C03575=1022.958,345.927,-141.680,171.455,48.856,159.616
C03576=1022.966,346.174,-141.717,171.462,48.856,159.617
C03577=1022.973,346.421,-141.753,171.468,48.855,159.618
C03578=1022.981,346.668,-141.790,171.475,48.854,159.618
C03579=1022.989,346.915,-141.828,171.483,48.853,159.619
C03580=1022.997,347.162,-141.865,171.489,48.852,159.620
C03581=1023.003,347.410,-141.902,171.496,48.851,159.621
C03582=1023.011,347.657,-141.939,171.502,48.850,159.622
C03583=1023.019,347.904,-141.976,171.510,48.849,159.623
C03584=1023.027,348.151,-142.013,171.517,48.848,159.623
C03585=1023.034,348.398,-142.051,171.524,48.848,159.624
C03586=1023.042,348.645,-142.087,171.530,48.847,159.625
C03587=1023.050,348.892,-142.125,171.538,48.846,159.626
C03588=1023.057,349.140,-142.163,171.545,48.845,159.627
C03589=1023.065,349.386,-142.200,171.551,48.845,159.628
C03590=1023.072,349.634,-142.237,171.559,48.844,159.629
C03591=1023.079,349.881,-142.275,171.566,48.843,159.629
C03592=1023.087,350.127,-142.312,171.573,48.843,159.630
C03593=1023.095,350.375,-142.349,171.580,48.842,159.631
C03594=1023.103,350.622,-142.387,171.587,48.841,159.632
C03595=1023.110,350.869,-142.424,171.594,48.840,159.633
C03596=1023.117,351.103,-142.460,171.601,48.840,159.634
C03597=1023.125,351.336,-142.495,171.607,48.839,159.635
C03598=1023.132,351.570,-142.532,171.614,48.838,159.635
C03599=1023.139,351.803,-142.567,171.621,48.838,159.636
C03600=1023.147,352.037,-142.602,171.628,48.838,159.637
C03601=1023.154,352.271,-142.638,171.635,48.837,159.638
C03602=1023.161,352.504,-142.673,171.641,48.836,159.639
C03603=1023.169,352.738,-142.709,171.648,48.836,159.640
C03604=1023.176,352.984,-142.747,171.656,48.835,159.641
C03605=1023.185,353.232,-142.784,171.662,48.834,159.642
C03606=1023.192,353.479,-142.822,171.669,48.834,159.643
C03607=1023.200,353.725,-142.860,171.677,48.833,159.644
C03608=1023.208,353.973,-142.897,171.684,48.832,159.644
C03609=1023.216,354.219,-142.935,171.692,48.832,159.646
C03610=1023.224,354.467,-142.973,171.699,48.831,159.646
C03611=1023.231,354.714,-143.012,171.707,48.831,159.648
C03612=1023.240,354.960,-143.049,171.714,48.830,159.648
C03613=1023.247,355.208,-143.087,171.721,48.830,159.649
C03614=1023.255,355.454,-143.125,171.728,48.829,159.650
C03615=1023.263,355.701,-143.164,171.735,48.829,159.651
C03616=1023.270,355.949,-143.201,171.743,48.828,159.652
C03617=1023.278,356.196,-143.240,171.750,48.828,159.653
C03618=1023.287,356.442,-143.278,171.758,48.827,159.654
C03619=1023.295,356.690,-143.316,171.765,48.827,159.655
C03620=1023.302,356.936,-143.354,171.773,48.827,159.656
C03621=1023.310,357.184,-143.392,171.780,48.826,159.657
C03622=1023.318,357.430,-143.431,171.788,48.826,159.658
C03623=1023.326,357.677,-143.469,171.795,48.825,159.659
C03624=1023.334,357.924,-143.508,171.803,48.824,159.660
C03625=1023.342,358.171,-143.546,171.810,48.824,159.661
C03626=1023.350,358.417,-143.584,171.818,48.824,159.663
C03627=1023.358,358.664,-143.622,171.825,48.824,159.664
C03628=1023.366,358.912,-143.661,171.833,48.824,159.665
C03629=1023.374,359.158,-143.699,171.840,48.823,159.666
C03630=1023.382,359.405,-143.738,171.848,48.823,159.667
C03631=1023.390,359.653,-143.776,171.855,48.823,159.668
C03632=1023.398,359.899,-143.815,171.863,48.822,159.669
C03633=1023.406,360.146,-143.853,171.870,48.822,159.670
C03634=1023.414,360.394,-143.892,171.878,48.822,159.671
C03635=1023.422,360.639,-143.931,171.885,48.822,159.672
C03636=1023.429,360.887,-143.970,171.893,48.821,159.673
C03637=1023.437,361.134,-144.009,171.900,48.821,159.674
C03638=1023.445,361.380,-144.048,171.908,48.821,159.675
C03639=1023.453,361.627,-144.086,171.916,48.820,159.676
C03640=1023.462,361.874,-144.126,171.924,48.820,159.677
C03641=1023.470,362.121,-144.164,171.932,48.821,159.679
C03642=1023.477,362.367,-144.204,171.939,48.821,159.680
C03643=1023.485,362.615,-144.242,171.947,48.820,159.681
C03644=1023.494,362.861,-144.282,171.955,48.820,159.682
C03645=1023.502,363.108,-144.320,171.963,48.820,159.683
C03646=1023.510,363.355,-144.360,171.971,48.820,159.684
C03647=1023.517,363.602,-144.398,171.978,48.820,159.685
C03648=1023.526,363.848,-144.438,171.986,48.819,159.687
C03649=1023.534,364.095,-144.477,171.994,48.820,159.688
C03650=1023.542,364.342,-144.516,172.001,48.820,159.689
C03651=1023.551,364.589,-144.555,172.009,48.819,159.690
C03652=1023.558,364.836,-144.595,172.018,48.819,159.691
C03653=1023.567,365.083,-144.634,172.025,48.819,159.692
C03654=1023.575,365.330,-144.673,172.033,48.820,159.694
C03655=1023.583,365.576,-144.712,172.041,48.819,159.695
C03656=1023.591,365.813,-144.750,172.049,48.819,159.696
C03657=1023.599,366.049,-144.788,172.057,48.819,159.697
C03658=1023.608,366.287,-144.825,172.064,48.819,159.698
C03659=1023.615,366.524,-144.863,172.072,48.819,159.700
C03660=1023.623,366.761,-144.901,172.080,48.819,159.701
C03661=1023.631,366.998,-144.940,172.088,48.820,159.702
C03662=1023.639,367.235,-144.977,172.095,48.820,159.703
C03663=1023.647,367.471,-145.015,172.103,48.819,159.704
C03664=1023.656,367.719,-145.055,172.111,48.820,159.705
C03665=1023.664,367.965,-145.094,172.119,48.820,159.707
C03666=1023.673,368.212,-145.134,172.127,48.819,159.708
C03667=1023.680,368.459,-145.174,172.135,48.820,159.709
C03668=1023.689,368.705,-145.213,172.144,48.820,159.710
C03669=1023.697,368.952,-145.253,172.151,48.820,159.712
C03670=1023.705,369.198,-145.293,172.160,48.821,159.713
C03671=1023.713,369.445,-145.333,172.168,48.821,159.714
C03672=1023.722,369.693,-145.372,172.177,48.821,159.716
C03673=1023.730,369.939,-145.413,172.185,48.821,159.717
C03674=1023.739,370.185,-145.452,172.192,48.822,159.718
C03675=1023.747,370.432,-145.493,172.201,48.822,159.719
C03676=1023.755,370.678,-145.532,172.209,48.822,159.721
C03677=1023.764,370.925,-145.573,172.218,48.822,159.722
C03678=1023.772,371.172,-145.613,172.226,48.823,159.723
C03679=1023.780,371.418,-145.653,172.235,48.823,159.725
C03680=1023.789,371.665,-145.693,172.243,48.823,159.726
C03681=1023.797,371.912,-145.734,172.250,48.824,159.727
C03682=1023.806,372.158,-145.774,172.259,48.824,159.729
C03683=1023.814,372.405,-145.814,172.267,48.824,159.730
C03684=1023.822,372.652,-145.855,172.276,48.825,159.731
C03685=1023.831,372.898,-145.895,172.284,48.825,159.733
C03686=1023.839,373.145,-145.935,172.293,48.825,159.734
C03687=1023.848,373.391,-145.975,172.301,48.825,159.735
C03688=1023.856,373.637,-146.016,172.310,48.826,159.737
C03689=1023.866,373.884,-146.056,172.319,48.826,159.738
C03690=1023.874,374.130,-146.097,172.327,48.826,159.740
C03691=1023.883,374.377,-146.137,172.336,48.827,159.741
C03692=1023.891,374.623,-146.178,172.344,48.827,159.742
C03693=1023.900,374.870,-146.218,172.353,48.828,159.744
C03694=1023.908,375.117,-146.258,172.361,48.828,159.745
C03695=1023.917,375.364,-146.298,172.370,48.829,159.747
C03696=1023.926,375.609,-146.340,172.379,48.829,159.748
C03697=1023.935,375.856,-146.380,172.387,48.830,159.750
C03698=1023.943,376.102,-146.421,172.396,48.830,159.751
C03699=1023.952,376.349,-146.462,172.405,48.831,159.752
C03700=1023.961,376.596,-146.502,172.413,48.831,159.754
C03701=1023.969,376.842,-146.543,172.422,48.832,159.755
C03702=1023.978,377.089,-146.585,172.431,48.833,159.757
C03703=1023.987,377.336,-146.626,172.439,48.833,159.758
C03704=1023.995,377.582,-146.666,172.448,48.834,159.760
C03705=1024.004,377.828,-146.707,172.457,48.835,159.761
C03706=1024.013,378.074,-146.748,172.466,48.835,159.763
C03707=1024.021,378.320,-146.790,172.475,48.836,159.764
C03708=1024.030,378.567,-146.831,172.484,48.837,159.766
C03709=1024.038,378.813,-146.872,172.493,48.838,159.767
C03710=1024.047,379.060,-146.913,172.501,48.838,159.769
C03711=1024.056,379.306,-146.955,172.510,48.839,159.770
C03712=1024.065,379.553,-146.997,172.519,48.840,159.772
C03713=1024.073,379.799,-147.037,172.528,48.841,159.773
C03714=1024.083,380.045,-147.078,172.538,48.841,159.775
C03715=1024.092,380.292,-147.120,172.546,48.842,159.776
C03716=1024.100,380.541,-147.162,172.555,48.843,159.778
C03717=1024.109,380.790,-147.203,172.564,48.843,159.779
C03718=1024.118,381.039,-147.246,172.574,48.844,159.781
C03719=1024.127,381.288,-147.287,172.583,48.845,159.783
C03720=1024.136,381.535,-147.329,172.592,48.846,159.784
C03721=1024.145,381.781,-147.371,172.601,48.846,159.786
C03722=1024.154,382.027,-147.412,172.610,48.847,159.787
C03723=1024.163,382.274,-147.454,172.619,48.849,159.789
C03724=1024.172,382.520,-147.496,172.628,48.849,159.791
C03725=1024.181,382.766,-147.537,172.638,48.850,159.792
C03726=1024.190,383.013,-147.579,172.647,48.851,159.794
C03727=1024.199,383.259,-147.620,172.656,48.852,159.795
C03728=1024.208,383.505,-147.662,172.666,48.852,159.797
C03729=1024.217,383.752,-147.704,172.675,48.854,159.799
C03730=1024.226,383.998,-147.745,172.684,48.854,159.800
C03731=1024.235,384.244,-147.788,172.694,48.855,159.802
C03732=1024.244,384.490,-147.830,172.702,48.856,159.804
C03733=1024.253,384.737,-147.871,172.713,48.857,159.805
C03734=1024.263,384.983,-147.913,172.722,48.859,159.807
C03735=1024.273,385.229,-147.955,172.730,48.859,159.809
C03736=1024.282,385.475,-147.997,172.741,48.860,159.810
C03737=1024.290,385.722,-148.039,172.749,48.861,159.812
C03738=1024.300,385.968,-148.081,172.760,48.862,159.814
C03739=1024.309,386.215,-148.123,172.769,48.863,159.816
C03740=1024.318,386.460,-148.166,172.779,48.864,159.817
C03741=1024.327,386.706,-148.209,172.788,48.866,159.819
C03742=1024.336,386.953,-148.250,172.797,48.867,159.821
C03743=1024.346,387.199,-148.293,172.807,48.868,159.822
C03744=1024.355,387.445,-148.336,172.816,48.869,159.824
C03745=1024.364,387.691,-148.377,172.826,48.870,159.826
C03746=1024.373,387.937,-148.420,172.835,48.871,159.828
C03747=1024.383,388.183,-148.463,172.845,48.872,159.829
C03748=1024.391,388.430,-148.506,172.856,48.873,159.831
C03749=1024.401,388.676,-148.548,172.865,48.875,159.833
C03750=1024.411,388.922,-148.591,172.875,48.876,159.835
C03751=1024.420,389.167,-148.633,172.884,48.877,159.837
C03752=1024.429,389.414,-148.677,172.894,48.878,159.838
C03753=1024.438,389.660,-148.719,172.904,48.880,159.840
C03754=1024.448,389.906,-148.762,172.914,48.881,159.842
C03755=1024.457,390.152,-148.804,172.924,48.882,159.844
C03756=1024.466,390.398,-148.847,172.933,48.884,159.846
C03757=1024.476,390.645,-148.890,172.944,48.885,159.848
C03758=1024.485,390.890,-148.933,172.954,48.886,159.849
C03759=1024.494,391.137,-148.977,172.963,48.888,159.851
C03760=1024.504,391.383,-149.019,172.974,48.889,159.853
C03761=1024.513,391.629,-149.062,172.984,48.890,159.855
C03762=1024.523,391.875,-149.106,172.993,48.892,159.857
C03763=1024.532,392.121,-149.148,173.003,48.893,159.859
C03764=1024.542,392.367,-149.191,173.014,48.895,159.861
C03765=1024.551,392.613,-149.235,173.023,48.897,159.863
C03766=1024.560,392.859,-149.278,173.034,48.897,159.864
C03767=1024.571,393.105,-149.321,173.044,48.899,159.866
C03768=1024.580,393.351,-149.365,173.055,48.901,159.869
C03769=1024.589,393.597,-149.408,173.065,48.902,159.870
C03770=1024.599,393.843,-149.452,173.074,48.903,159.872
C03771=1024.609,394.089,-149.495,173.085,48.905,159.874
C03772=1024.617,394.335,-149.538,173.095,48.907,159.876
C03773=1024.627,394.580,-149.582,173.106,48.908,159.878
C03774=1024.637,394.827,-149.626,173.116,48.910,159.880
C03775=1024.647,395.072,-149.670,173.126,48.912,159.882
C03776=1024.658,395.359,-149.720,173.139,48.913,159.885
C03777=1024.669,395.643,-149.771,173.150,48.915,159.887
C03778=1024.681,395.930,-149.821,173.162,48.917,159.889
C03779=1024.692,396.216,-149.873,173.174,48.919,159.892
C03780=1024.702,396.461,-149.917,173.185,48.921,159.894
C03781=1024.711,396.708,-149.961,173.195,48.922,159.896
C03782=1024.721,396.953,-150.004,173.206,48.924,159.898
C03783=1024.731,397.199,-150.048,173.216,48.925,159.900
C03784=1024.741,397.445,-150.093,173.227,48.927,159.902
C03785=1024.751,397.691,-150.137,173.238,48.929,159.904
C03786=1024.761,397.937,-150.180,173.248,48.931,159.906
C03787=1024.770,398.183,-150.224,173.259,48.933,159.908
C03788=1024.781,398.428,-150.269,173.270,48.934,159.910
C03789=1024.790,398.674,-150.313,173.281,48.936,159.912
C03790=1024.800,398.920,-150.357,173.291,48.938,159.914
C03791=1024.810,399.165,-150.401,173.302,48.940,159.917
C03792=1024.820,399.411,-150.446,173.312,48.941,159.919
C03793=1024.830,399.658,-150.490,173.324,48.943,159.921
C03794=1024.840,399.903,-150.534,173.335,48.945,159.923
C03795=1024.850,400.149,-150.579,173.346,48.947,159.925
C03796=1024.860,400.394,-150.624,173.357,48.949,159.927
C03797=1024.869,400.640,-150.668,173.367,48.951,159.929
C03798=1024.880,400.886,-150.713,173.378,48.953,159.932
C03799=1024.890,401.132,-150.758,173.389,48.955,159.934
C03800=1024.899,401.377,-150.802,173.401,48.956,159.936
C03801=1024.909,401.623,-150.847,173.411,48.959,159.938
C03802=1024.919,401.869,-150.892,173.422,48.961,159.940
C03803=1024.929,402.114,-150.937,173.433,48.963,159.943
C03804=1024.940,402.360,-150.982,173.445,48.964,159.945
C03805=1024.950,402.606,-151.027,173.456,48.967,159.947
C03806=1024.960,402.851,-151.072,173.467,48.969,159.950
C03807=1024.970,403.097,-151.117,173.478,48.971,159.952
C03808=1024.980,403.342,-151.162,173.490,48.973,159.954
C03809=1024.990,403.588,-151.207,173.501,48.975,159.956
C03810=1025.000,403.834,-151.252,173.512,48.978,159.959
C03811=1025.010,404.079,-151.298,173.524,48.980,159.961
C03812=1025.020,404.325,-151.343,173.535,48.982,159.963
C03813=1025.030,404.571,-151.388,173.547,48.984,159.966
C03814=1025.041,404.816,-151.434,173.558,48.986,159.968
C03815=1025.051,405.063,-151.479,173.569,48.988,159.970
C03816=1025.062,405.307,-151.524,173.581,48.990,159.973
C03817=1025.072,405.553,-151.569,173.592,48.992,159.975
C03818=1025.083,405.799,-151.615,173.604,48.995,159.977
C03819=1025.093,406.044,-151.661,173.615,48.997,159.980
C03820=1025.103,406.290,-151.706,173.627,48.999,159.982
C03821=1025.114,406.536,-151.752,173.638,49.002,159.985
C03822=1025.124,406.781,-151.798,173.651,49.004,159.987
C03823=1025.134,407.026,-151.843,173.662,49.006,159.989
C03824=1025.145,407.272,-151.888,173.674,49.008,159.992
C03825=1025.155,407.518,-151.934,173.686,49.011,159.994
C03826=1025.166,407.763,-151.980,173.697,49.013,159.997
C03827=1025.176,408.009,-152.026,173.709,49.016,159.999
C03828=1025.188,408.254,-152.071,173.722,49.018,160.002
C03829=1025.198,408.500,-152.117,173.733,49.020,160.004
C03830=1025.209,408.746,-152.163,173.745,49.023,160.007
C03831=1025.220,408.991,-152.209,173.757,49.025,160.009
C03832=1025.230,409.237,-152.255,173.770,49.027,160.012
C03833=1025.241,409.482,-152.301,173.781,49.030,160.014
C03834=1025.252,409.727,-152.347,173.793,49.032,160.017
C03835=1025.263,409.973,-152.393,173.806,49.035,160.019
C03836=1025.275,410.282,-152.452,173.821,49.038,160.022
C03837=1025.289,410.590,-152.511,173.836,49.041,160.026
C03838=1025.302,410.898,-152.568,173.851,49.044,160.029
C03839=1025.316,411.206,-152.627,173.867,49.048,160.032
C03840=1025.326,411.451,-152.673,173.879,49.050,160.035
C03841=1025.337,411.697,-152.721,173.891,49.053,160.037
C03842=1025.348,411.942,-152.767,173.904,49.056,160.040
C03843=1025.359,412.188,-152.813,173.916,49.058,160.043
C03844=1025.370,412.433,-152.860,173.929,49.061,160.045
C03845=1025.380,412.679,-152.907,173.941,49.063,160.048
C03846=1025.391,412.924,-152.954,173.954,49.066,160.051
C03847=1025.402,413.169,-153.001,173.966,49.068,160.053
C03848=1025.414,413.414,-153.048,173.979,49.071,160.056
C03849=1025.424,413.660,-153.095,173.992,49.074,160.059
C03850=1025.435,413.905,-153.141,174.004,49.077,160.062
C03851=1025.446,414.150,-153.188,174.017,49.080,160.064
C03852=1025.457,414.395,-153.235,174.029,49.082,160.067
C03853=1025.468,414.641,-153.283,174.042,49.085,160.070
C03854=1025.479,414.886,-153.329,174.055,49.088,160.072
C03855=1025.491,415.131,-153.377,174.069,49.091,160.075
C03856=1025.502,415.377,-153.424,174.081,49.094,160.078
C03857=1025.513,415.622,-153.471,174.094,49.097,160.081
C03858=1025.524,415.868,-153.518,174.106,49.099,160.084
C03859=1025.535,416.113,-153.566,174.119,49.103,160.087
C03860=1025.546,416.358,-153.613,174.133,49.105,160.089
C03861=1025.557,416.604,-153.661,174.146,49.108,160.092
C03862=1025.569,416.849,-153.709,174.159,49.111,160.095
C03863=1025.579,417.094,-153.756,174.173,49.114,160.098
C03864=1025.591,417.339,-153.804,174.185,49.117,160.101
C03865=1025.602,417.584,-153.852,174.198,49.120,160.104
C03866=1025.614,417.829,-153.900,174.212,49.123,160.107
C03867=1025.625,418.074,-153.948,174.225,49.127,160.110
C03868=1025.636,418.320,-153.995,174.238,49.129,160.112
C03869=1025.647,418.565,-154.043,174.252,49.132,160.115
C03870=1025.659,418.810,-154.091,174.265,49.136,160.118
C03871=1025.670,419.056,-154.139,174.279,49.139,160.121
C03872=1025.682,419.300,-154.188,174.292,49.142,160.124
C03873=1025.693,419.545,-154.236,174.306,49.145,160.127
C03874=1025.705,419.790,-154.284,174.320,49.148,160.130
C03875=1025.716,420.036,-154.332,174.333,49.151,160.133
C03876=1025.728,420.281,-154.380,174.347,49.155,160.136
C03877=1025.740,420.526,-154.429,174.360,49.158,160.139
C03878=1025.751,420.771,-154.476,174.374,49.161,160.142
C03879=1025.762,421.016,-154.525,174.388,49.164,160.145
C03880=1025.775,421.260,-154.573,174.401,49.167,160.149
C03881=1025.786,421.506,-154.621,174.415,49.170,160.152
C03882=1025.798,421.751,-154.670,174.430,49.174,160.155
C03883=1025.810,421.996,-154.718,174.444,49.177,160.158
C03884=1025.821,422.241,-154.767,174.458,49.180,160.161
C03885=1025.833,422.485,-154.816,174.471,49.184,160.164
C03886=1025.845,422.731,-154.865,174.485,49.187,160.167
C03887=1025.857,422.976,-154.914,174.500,49.190,160.170
C03888=1025.868,423.220,-154.963,174.514,49.194,160.174
C03889=1025.881,423.466,-155.012,174.528,49.197,160.177
C03890=1025.892,423.710,-155.061,174.542,49.200,160.180
C03891=1025.903,423.955,-155.110,174.557,49.204,160.183
C03892=1025.915,424.200,-155.159,174.571,49.207,160.186
C03893=1025.928,424.445,-155.208,174.585,49.211,160.190
C03894=1025.940,424.690,-155.257,174.600,49.215,160.193
C03895=1025.951,424.935,-155.306,174.615,49.218,160.196
C03896=1025.967,425.254,-155.371,174.633,49.223,160.201
C03897=1025.982,425.573,-155.435,174.652,49.227,160.205
C03898=1025.998,425.892,-155.499,174.671,49.232,160.209
C03899=1026.014,426.211,-155.563,174.691,49.236,160.214
C03900=1026.027,426.455,-155.613,174.706,49.240,160.217
C03901=1026.039,426.701,-155.663,174.720,49.244,160.220
C03902=1026.050,426.945,-155.713,174.735,49.248,160.224
C03903=1026.063,427.190,-155.763,174.750,49.251,160.227
C03904=1026.075,427.435,-155.813,174.765,49.255,160.230
C03905=1026.087,427.679,-155.863,174.780,49.259,160.234
C03906=1026.099,427.924,-155.913,174.795,49.262,160.237
C03907=1026.111,428.168,-155.963,174.810,49.266,160.241
C03908=1026.124,428.413,-156.013,174.825,49.270,160.244
C03909=1026.136,428.658,-156.063,174.840,49.274,160.248
C03910=1026.148,428.903,-156.113,174.855,49.278,160.251
C03911=1026.160,429.148,-156.163,174.871,49.281,160.255
C03912=1026.173,429.393,-156.213,174.886,49.285,160.258
C03913=1026.185,429.637,-156.264,174.901,49.289,160.262
C03914=1026.198,429.882,-156.314,174.918,49.293,160.266
C03915=1026.210,430.126,-156.365,174.932,49.297,160.269
C03916=1026.223,430.371,-156.415,174.948,49.300,160.273
C03917=1026.235,430.615,-156.465,174.963,49.305,160.276
C03918=1026.248,430.860,-156.516,174.979,49.308,160.280
C03919=1026.261,431.105,-156.567,174.995,49.312,160.284
C03920=1026.273,431.349,-156.617,175.011,49.316,160.287
C03921=1026.286,431.594,-156.668,175.027,49.320,160.291
C03922=1026.298,431.838,-156.719,175.042,49.324,160.294
C03923=1026.312,432.083,-156.770,175.058,49.329,160.298
C03924=1026.324,432.327,-156.820,175.074,49.333,160.302
C03925=1026.337,432.572,-156.871,175.090,49.337,160.306
C03926=1026.350,432.817,-156.922,175.107,49.341,160.309
C03927=1026.363,433.061,-156.973,175.123,49.345,160.313
C03928=1026.376,433.306,-157.024,175.139,49.349,160.317
C03929=1026.389,433.550,-157.076,175.155,49.353,160.321
C03930=1026.402,433.794,-157.127,175.171,49.357,160.324
C03931=1026.414,434.038,-157.178,175.188,49.361,160.328
C03932=1026.428,434.283,-157.229,175.204,49.365,160.332
C03933=1026.441,434.528,-157.281,175.220,49.370,160.336
C03934=1026.453,434.771,-157.333,175.237,49.374,160.340
C03935=1026.466,435.016,-157.384,175.254,49.378,160.344
C03936=1026.480,435.261,-157.436,175.270,49.382,160.348
C03937=1026.493,435.505,-157.487,175.287,49.387,160.352
C03938=1026.506,435.749,-157.538,175.304,49.391,160.356
C03939=1026.519,435.994,-157.591,175.321,49.396,160.360
C03940=1026.532,436.237,-157.643,175.337,49.400,160.363
C03941=1026.545,436.482,-157.694,175.354,49.404,160.367
C03942=1026.559,436.726,-157.746,175.371,49.408,160.371
C03943=1026.572,436.970,-157.799,175.389,49.413,160.376
C03944=1026.585,437.215,-157.851,175.405,49.417,160.380
C03945=1026.599,437.459,-157.903,175.423,49.422,160.384
C03946=1026.612,437.703,-157.954,175.439,49.426,160.388
C03947=1026.625,437.947,-158.008,175.457,49.431,160.392
C03948=1026.639,438.192,-158.060,175.475,49.435,160.396
C03949=1026.652,438.436,-158.111,175.491,49.439,160.400
C03950=1026.666,438.680,-158.165,175.509,49.444,160.404
C03951=1026.679,438.924,-158.217,175.527,49.449,160.409
C03952=1026.693,439.168,-158.269,175.543,49.453,160.413
C03953=1026.706,439.412,-158.322,175.561,49.458,160.417
C03954=1026.720,439.656,-158.374,175.579,49.462,160.421
C03955=1026.734,439.900,-158.427,175.597,49.467,160.425
C03956=1026.747,440.144,-158.480,175.615,49.472,160.430
C03957=1026.760,440.390,-158.533,175.633,49.476,160.434
C03958=1026.775,440.634,-158.586,175.651,49.481,160.438
C03959=1026.789,440.879,-158.640,175.669,49.486,160.442
C03960=1026.801,441.107,-158.689,175.686,49.490,160.447
C03961=1026.815,441.334,-158.738,175.703,49.495,160.451
C03962=1026.828,441.561,-158.788,175.720,49.499,160.455
C03963=1026.840,441.790,-158.838,175.736,49.503,160.459
C03964=1026.853,442.017,-158.888,175.754,49.508,160.463
C03965=1026.867,442.244,-158.937,175.771,49.512,160.467
C03966=1026.880,442.472,-158.987,175.789,49.517,160.471
C03967=1026.893,442.700,-159.036,175.805,49.521,160.475
C03968=1026.908,442.942,-159.089,175.823,49.526,160.480
C03969=1026.922,443.185,-159.142,175.842,49.530,160.484
C03970=1026.938,443.429,-159.194,175.862,49.535,160.489
C03971=1026.954,443.673,-159.245,175.879,49.540,160.493
C03972=1026.971,443.916,-159.297,175.899,49.544,160.497
C03973=1026.987,444.160,-159.347,175.918,49.548,160.502
C03974=1027.005,444.403,-159.398,175.937,49.553,160.506
C03975=1027.022,444.648,-159.448,175.956,49.557,160.511
C03976=1027.041,444.892,-159.498,175.975,49.561,160.515
C03977=1027.060,445.136,-159.547,175.994,49.565,160.519
C03978=1027.079,445.380,-159.595,176.013,49.569,160.524
C03979=1027.098,445.624,-159.644,176.033,49.573,160.528
C03980=1027.118,445.869,-159.692,176.052,49.577,160.532
C03981=1027.138,446.113,-159.739,176.072,49.581,160.537
C03982=1027.159,446.357,-159.787,176.092,49.585,160.541
C03983=1027.181,446.601,-159.834,176.112,49.588,160.545
C03984=1027.203,446.845,-159.881,176.132,49.592,160.550
C03985=1027.225,447.091,-159.927,176.151,49.596,160.554
C03986=1027.248,447.335,-159.972,176.172,49.599,160.559
C03987=1027.272,447.580,-160.017,176.192,49.603,160.563
C03988=1027.295,447.825,-160.062,176.212,49.606,160.567
C03989=1027.319,448.069,-160.107,176.232,49.609,160.571
C03990=1027.345,448.315,-160.151,176.253,49.612,160.576
C03991=1027.369,448.559,-160.195,176.274,49.615,160.580
C03992=1027.395,448.804,-160.239,176.295,49.619,160.585
C03993=1027.421,449.049,-160.281,176.315,49.621,160.589
C03994=1027.447,449.295,-160.323,176.336,49.624,160.593
C03995=1027.475,449.539,-160.365,176.357,49.628,160.597
C03996=1027.502,449.785,-160.407,176.377,49.630,160.602
C03997=1027.530,450.030,-160.449,176.399,49.633,160.606
C03998=1027.559,450.275,-160.490,176.419,49.636,160.610
C03999=1027.587,450.521,-160.531,176.441,49.638,160.615
C04000=1027.617,450.766,-160.571,176.462,49.641,160.619
C04001=1027.646,451.012,-160.611,176.483,49.644,160.623
C04002=1027.677,451.257,-160.650,176.504,49.647,160.628
C04003=1027.707,451.502,-160.689,176.526,49.649,160.632
C04004=1027.738,451.748,-160.728,176.548,49.651,160.636
C04005=1027.771,451.994,-160.765,176.570,49.653,160.640
C04006=1027.802,452.240,-160.804,176.591,49.656,160.645
C04007=1027.835,452.485,-160.841,176.614,49.658,160.649
C04008=1027.868,452.731,-160.878,176.635,49.660,160.653
C04009=1027.902,452.977,-160.914,176.658,49.662,160.658
C04010=1027.935,453.222,-160.950,176.680,49.664,160.662
C04011=1027.971,453.468,-160.987,176.703,49.666,160.666
C04012=1028.005,453.714,-161.021,176.725,49.668,160.671
C04013=1028.040,453.960,-161.057,176.747,49.670,160.675
C04014=1028.076,454.206,-161.091,176.770,49.672,160.679
C04015=1028.113,454.451,-161.125,176.792,49.674,160.683
C04016=1027.838,454.527,-161.463,176.795,49.734,160.703
C04017=1027.801,454.282,-161.428,176.773,49.732,160.699
C04018=1027.765,454.036,-161.394,176.749,49.731,160.694
C04019=1027.730,453.790,-161.359,176.727,49.729,160.690
C04020=1027.695,453.544,-161.324,176.705,49.727,160.686
C04021=1027.660,453.298,-161.289,176.682,49.725,160.681
C04022=1027.626,453.053,-161.252,176.660,49.723,160.677
C04023=1027.593,452.807,-161.215,176.638,49.722,160.673
C04024=1027.560,452.561,-161.179,176.616,49.719,160.669
C04025=1027.527,452.316,-161.142,176.594,49.717,160.664
C04026=1027.494,452.070,-161.104,176.572,49.715,160.660
C04027=1027.463,451.824,-161.066,176.550,49.713,160.656
C04028=1027.431,451.578,-161.028,176.528,49.711,160.652
C04029=1027.400,451.334,-160.988,176.506,49.708,160.647
C04030=1027.370,451.088,-160.950,176.485,49.706,160.643
C04031=1027.340,450.842,-160.910,176.463,49.703,160.639
C04032=1027.310,450.596,-160.870,176.442,49.701,160.634
C04033=1027.281,450.351,-160.829,176.421,49.699,160.630
C04034=1027.253,450.106,-160.789,176.400,49.695,160.626
C04035=1027.224,449.861,-160.748,176.378,49.693,160.621
C04036=1027.197,449.616,-160.706,176.358,49.690,160.617
C04037=1027.170,449.370,-160.664,176.336,49.687,160.613
C04038=1027.143,449.126,-160.622,176.316,49.685,160.609
C04039=1027.117,448.880,-160.579,176.295,49.681,160.604
C04040=1027.091,448.635,-160.535,176.274,49.679,160.600
C04041=1027.065,448.390,-160.492,176.254,49.676,160.596
C04042=1027.041,448.145,-160.449,176.233,49.672,160.591
C04043=1027.016,447.900,-160.404,176.213,49.670,160.587
C04044=1026.992,447.656,-160.359,176.193,49.666,160.583
C04045=1026.969,447.411,-160.314,176.172,49.663,160.578
C04046=1026.945,447.166,-160.268,176.152,49.659,160.574
C04047=1026.923,446.921,-160.223,176.132,49.656,160.570
C04048=1026.902,446.677,-160.176,176.112,49.653,160.565
C04049=1026.880,446.432,-160.129,176.092,49.649,160.561
C04050=1026.858,446.187,-160.082,176.072,49.646,160.557
C04051=1026.838,445.944,-160.035,176.052,49.642,160.552
C04052=1026.817,445.699,-159.987,176.033,49.638,160.548
C04053=1026.798,445.455,-159.939,176.013,49.634,160.544
C04054=1026.778,445.210,-159.890,175.994,49.630,160.539
C04055=1026.759,444.967,-159.841,175.975,49.626,160.535
C04056=1026.741,444.723,-159.791,175.956,49.622,160.531
C04057=1026.723,444.479,-159.742,175.936,49.618,160.526
C04058=1026.705,444.234,-159.692,175.917,49.614,160.522
C04059=1026.688,443.991,-159.641,175.898,49.610,160.517
C04060=1026.671,443.748,-159.590,175.879,49.606,160.513
C04061=1026.655,443.503,-159.539,175.860,49.601,160.508
C04062=1026.639,443.260,-159.486,175.842,49.597,160.504
C04063=1026.625,443.017,-159.434,175.823,49.592,160.500
C04064=1026.610,442.774,-159.381,175.804,49.587,160.495
C04065=1026.595,442.531,-159.329,175.786,49.583,160.491
C04066=1026.581,442.287,-159.275,175.767,49.578,160.486
C04067=1026.567,442.043,-159.223,175.749,49.573,160.482
C04068=1026.553,441.800,-159.169,175.730,49.569,160.478
C04069=1026.540,441.576,-159.121,175.714,49.565,160.474
C04070=1026.527,441.353,-159.072,175.697,49.561,160.470
C04071=1026.515,441.129,-159.024,175.681,49.556,160.466
C04072=1026.502,440.905,-158.975,175.664,49.552,160.462
C04073=1026.489,440.681,-158.926,175.648,49.547,160.458
C04074=1026.477,440.458,-158.877,175.630,49.544,160.454
C04075=1026.464,440.234,-158.829,175.614,49.540,160.450
C04076=1026.452,440.011,-158.781,175.597,49.535,160.446
C04077=1026.438,439.766,-158.727,175.580,49.531,160.442
C04078=1026.424,439.522,-158.675,175.563,49.526,160.438
C04079=1026.411,439.278,-158.623,175.545,49.521,160.433
C04080=1026.397,439.034,-158.570,175.527,49.517,160.429
C04081=1026.384,438.790,-158.517,175.509,49.513,160.425
C04082=1026.370,438.546,-158.465,175.492,49.508,160.421
C04083=1026.357,438.302,-158.412,175.474,49.504,160.417
C04084=1026.343,438.057,-158.360,175.457,49.499,160.413
C04085=1026.329,437.813,-158.308,175.440,49.495,160.408
C04086=1026.316,437.569,-158.256,175.422,49.491,160.404
C04087=1026.303,437.325,-158.203,175.405,49.486,160.400
C04088=1026.290,437.081,-158.151,175.388,49.482,160.396
C04089=1026.276,436.837,-158.099,175.371,49.478,160.392
C04090=1026.263,436.592,-158.047,175.354,49.473,160.388
C04091=1026.249,436.348,-157.996,175.337,49.469,160.384
C04092=1026.236,436.104,-157.943,175.320,49.465,160.380
C04093=1026.219,435.783,-157.875,175.298,49.459,160.375
C04094=1026.202,435.462,-157.807,175.276,49.454,160.370
C04095=1026.184,435.142,-157.740,175.254,49.449,160.365
C04096=1026.168,434.821,-157.673,175.233,49.443,160.360
C04097=1026.154,434.577,-157.621,175.215,49.439,160.356
C04098=1026.142,434.332,-157.569,175.199,49.435,160.352
C04099=1026.129,434.088,-157.517,175.183,49.431,160.348
C04100=1026.116,433.843,-157.466,175.166,49.426,160.344
C04101=1026.103,433.599,-157.415,175.150,49.422,160.340
C04102=1026.089,433.355,-157.364,175.134,49.418,160.337
C04103=1026.077,433.111,-157.313,175.117,49.414,160.333
C04104=1026.064,432.866,-157.262,175.101,49.410,160.329
C04105=1026.051,432.621,-157.211,175.085,49.406,160.325
C04106=1026.038,432.377,-157.160,175.069,49.402,160.322
C04107=1026.025,432.132,-157.109,175.053,49.399,160.318
C04108=1026.013,431.888,-157.059,175.038,49.394,160.314
C04109=1026.000,431.643,-157.008,175.021,49.390,160.311
C04110=1025.988,431.399,-156.957,175.006,49.387,160.307
C04111=1025.974,431.154,-156.906,174.990,49.383,160.303
C04112=1025.962,430.909,-156.856,174.974,49.379,160.300
C04113=1025.949,430.665,-156.805,174.958,49.375,160.296
C04114=1025.937,430.420,-156.755,174.943,49.371,160.292
C04115=1025.924,430.176,-156.704,174.927,49.368,160.289
C04116=1025.912,429.931,-156.654,174.911,49.364,160.285
C04117=1025.900,429.687,-156.604,174.896,49.360,160.282
C04118=1025.887,429.442,-156.553,174.880,49.356,160.278
C04119=1025.875,429.198,-156.503,174.865,49.353,160.275
C04120=1025.863,428.953,-156.453,174.850,49.349,160.271
C04121=1025.850,428.708,-156.403,174.834,49.345,160.268
C04122=1025.837,428.464,-156.353,174.819,49.341,160.264
C04123=1025.825,428.219,-156.302,174.804,49.338,160.261
C04124=1025.812,427.974,-156.252,174.789,49.334,160.257
C04125=1025.800,427.730,-156.202,174.773,49.330,160.254
C04126=1025.788,427.484,-156.153,174.759,49.327,160.250
C04127=1025.776,427.240,-156.103,174.743,49.323,160.247
C04128=1025.764,426.995,-156.053,174.729,49.320,160.244
C04129=1025.752,426.750,-156.003,174.714,49.316,160.240
C04130=1025.740,426.506,-155.953,174.699,49.312,160.237
C04131=1025.728,426.261,-155.904,174.684,49.309,160.233
C04132=1025.716,426.016,-155.854,174.669,49.305,160.230
C04133=1025.704,425.770,-155.804,174.654,49.302,160.227
C04134=1025.692,425.526,-155.755,174.640,49.298,160.223
C04135=1025.679,425.281,-155.706,174.625,49.295,160.220
C04136=1025.667,425.036,-155.656,174.610,49.292,160.217
C04137=1025.656,424.791,-155.607,174.596,49.288,160.214
C04138=1025.643,424.546,-155.557,174.582,49.285,160.210
C04139=1025.631,424.302,-155.509,174.567,49.281,160.207
C04140=1025.619,424.056,-155.460,174.553,49.278,160.204
C04141=1025.608,423.812,-155.411,174.538,49.274,160.201
C04142=1025.596,423.567,-155.362,174.524,49.271,160.197
C04143=1025.584,423.322,-155.313,174.510,49.268,160.194
C04144=1025.572,423.077,-155.264,174.496,49.265,160.191
C04145=1025.561,422.832,-155.215,174.481,49.261,160.188
C04146=1025.548,422.587,-155.166,174.467,49.258,160.185
C04147=1025.537,422.342,-155.118,174.453,49.255,160.182
C04148=1025.526,422.097,-155.069,174.439,49.251,160.178
C04149=1025.514,421.852,-155.020,174.425,49.249,160.175
C04150=1025.502,421.607,-154.972,174.411,49.245,160.172
C04151=1025.490,421.362,-154.923,174.397,49.242,160.169
C04152=1025.479,421.117,-154.875,174.383,49.239,160.166
C04153=1025.467,420.872,-154.826,174.369,49.235,160.163
C04154=1025.455,420.626,-154.778,174.356,49.232,160.160
C04155=1025.444,420.381,-154.729,174.342,49.229,160.157
C04156=1025.431,420.136,-154.681,174.328,49.226,160.154
C04157=1025.420,419.891,-154.633,174.314,49.223,160.151
C04158=1025.409,419.646,-154.585,174.301,49.220,160.148
C04159=1025.397,419.401,-154.537,174.287,49.217,160.145
C04160=1025.386,419.156,-154.489,174.274,49.214,160.142
C04161=1025.375,418.910,-154.441,174.260,49.211,160.139
C04162=1025.363,418.666,-154.393,174.246,49.208,160.136
C04163=1025.352,418.421,-154.345,174.233,49.205,160.133
C04164=1025.340,418.175,-154.297,174.219,49.202,160.130
C04165=1025.329,417.930,-154.249,174.206,49.199,160.127
C04166=1025.317,417.685,-154.201,174.193,49.196,160.124
C04167=1025.306,417.440,-154.153,174.179,49.193,160.121
C04168=1025.295,417.195,-154.106,174.166,49.190,160.118
C04169=1025.284,416.949,-154.058,174.153,49.188,160.116
C04170=1025.272,416.704,-154.010,174.140,49.184,160.113
C04171=1025.262,416.459,-153.963,174.127,49.182,160.110
C04172=1025.250,416.214,-153.916,174.114,49.179,160.107
C04173=1025.239,415.969,-153.867,174.101,49.176,160.104
C04174=1025.228,415.724,-153.821,174.088,49.173,160.101
C04175=1025.218,415.478,-153.773,174.074,49.171,160.099
C04176=1025.206,415.233,-153.725,174.062,49.168,160.096
C04177=1025.195,414.988,-153.679,174.049,49.165,160.093
C04178=1025.183,414.742,-153.632,174.036,49.162,160.090
C04179=1025.173,414.497,-153.585,174.023,49.160,160.088
C04180=1025.162,414.251,-153.538,174.010,49.157,160.085
C04181=1025.151,414.006,-153.491,173.998,49.154,160.082
C04182=1025.139,413.760,-153.444,173.985,49.152,160.079
C04183=1025.129,413.515,-153.397,173.972,49.149,160.077
C04184=1025.117,413.269,-153.350,173.960,49.146,160.074
C04185=1025.106,413.024,-153.303,173.947,49.144,160.071
C04186=1025.096,412.779,-153.256,173.935,49.141,160.069
C04187=1025.085,412.533,-153.209,173.922,49.138,160.066
C04188=1025.074,412.288,-153.162,173.910,49.136,160.063
C04189=1025.063,412.043,-153.116,173.897,49.133,160.061
C04190=1025.052,411.798,-153.070,173.885,49.130,160.058
C04191=1025.042,411.553,-153.023,173.872,49.128,160.055
C04192=1025.031,411.307,-152.976,173.860,49.125,160.053
C04193=1025.018,410.997,-152.917,173.844,49.123,160.050
C04194=1025.004,410.686,-152.859,173.829,49.120,160.046
C04195=1024.990,410.375,-152.799,173.813,49.116,160.043
C04196=1024.977,410.065,-152.741,173.798,49.113,160.040
C04197=1024.966,409.820,-152.694,173.786,49.111,160.037
C04198=1024.955,409.575,-152.648,173.773,49.109,160.035
C04199=1024.945,409.329,-152.603,173.761,49.106,160.032
C04200=1024.934,409.083,-152.557,173.750,49.104,160.030
C04201=1024.924,408.838,-152.511,173.738,49.101,160.027
C04202=1024.913,408.592,-152.465,173.725,49.099,160.025
C04203=1024.902,408.347,-152.419,173.713,49.097,160.022
C04204=1024.892,408.101,-152.373,173.701,49.095,160.020
C04205=1024.881,407.855,-152.327,173.690,49.092,160.017
C04206=1024.870,407.610,-152.281,173.677,49.090,160.015
C04207=1024.860,407.364,-152.235,173.666,49.088,160.012
C04208=1024.849,407.119,-152.189,173.654,49.085,160.010
C04209=1024.839,406.873,-152.144,173.642,49.083,160.007
C04210=1024.828,406.628,-152.099,173.630,49.081,160.005
C04211=1024.817,406.382,-152.053,173.619,49.079,160.003
C04212=1024.807,406.137,-152.007,173.607,49.077,160.000
C04213=1024.797,405.890,-151.962,173.596,49.075,159.998
C04214=1024.787,405.645,-151.917,173.584,49.073,159.996
C04215=1024.776,405.400,-151.871,173.573,49.070,159.993
C04216=1024.766,405.154,-151.826,173.561,49.068,159.991
C04217=1024.756,404.909,-151.780,173.549,49.066,159.988
C04218=1024.745,404.663,-151.735,173.538,49.064,159.986
C04219=1024.736,404.417,-151.690,173.527,49.062,159.984
C04220=1024.725,404.171,-151.644,173.514,49.060,159.981
C04221=1024.714,403.926,-151.600,173.504,49.058,159.979
C04222=1024.704,403.680,-151.555,173.492,49.056,159.977
C04223=1024.694,403.435,-151.509,173.481,49.054,159.975
C04224=1024.684,403.189,-151.464,173.470,49.052,159.972
C04225=1024.674,402.943,-151.419,173.458,49.050,159.970
C04226=1024.664,402.697,-151.374,173.447,49.048,159.968
C04227=1024.654,402.452,-151.328,173.436,49.046,159.966
C04228=1024.644,402.207,-151.284,173.424,49.044,159.963
C04229=1024.634,401.961,-151.238,173.414,49.042,159.961
C04230=1024.624,401.715,-151.194,173.403,49.040,159.959
C04231=1024.614,401.470,-151.149,173.391,49.038,159.957
C04232=1024.604,401.224,-151.105,173.380,49.036,159.954
C04233=1024.594,400.978,-151.060,173.369,49.034,159.952
C04234=1024.584,400.732,-151.015,173.358,49.032,159.950
C04235=1024.574,400.487,-150.971,173.347,49.031,159.948
C04236=1024.564,400.241,-150.926,173.336,49.029,159.946
C04237=1024.554,399.994,-150.882,173.325,49.027,159.944
C04238=1024.544,399.749,-150.837,173.314,49.025,159.941
C04239=1024.534,399.504,-150.793,173.303,49.023,159.939
C04240=1024.524,399.258,-150.749,173.292,49.022,159.937
C04241=1024.515,399.012,-150.704,173.281,49.020,159.935
C04242=1024.504,398.766,-150.660,173.271,49.018,159.933
C04243=1024.495,398.521,-150.615,173.260,49.017,159.931
C04244=1024.485,398.275,-150.572,173.249,49.015,159.929
C04245=1024.474,398.029,-150.527,173.239,49.013,159.927
C04246=1024.465,397.783,-150.483,173.228,49.012,159.924
C04247=1024.455,397.537,-150.439,173.217,49.010,159.922
C04248=1024.445,397.291,-150.395,173.207,49.008,159.920
C04249=1024.435,397.045,-150.352,173.196,49.006,159.918
C04250=1024.425,396.799,-150.307,173.186,49.005,159.916
C04251=1024.415,396.553,-150.263,173.175,49.003,159.914
C04252=1024.407,396.308,-150.219,173.165,49.002,159.912
C04253=1024.395,396.019,-150.168,173.151,49.000,159.910
C04254=1024.383,395.732,-150.117,173.140,48.998,159.907
C04255=1024.372,395.444,-150.066,173.127,48.997,159.905
C04256=1024.361,395.155,-150.015,173.115,48.995,159.903
C04257=1024.351,394.909,-149.971,173.104,48.993,159.901
C04258=1024.341,394.663,-149.927,173.094,48.992,159.899
C04259=1024.332,394.418,-149.884,173.083,48.990,159.897
C04260=1024.322,394.172,-149.840,173.074,48.989,159.895
C04261=1024.312,393.925,-149.797,173.064,48.987,159.893
C04262=1024.303,393.679,-149.753,173.053,48.986,159.891
C04263=1024.294,393.434,-149.710,173.043,48.984,159.889
C04264=1024.284,393.187,-149.666,173.032,48.983,159.887
C04265=1024.274,392.942,-149.623,173.022,48.982,159.885
C04266=1024.265,392.696,-149.581,173.013,48.980,159.883
C04267=1024.256,392.450,-149.536,173.002,48.979,159.881
C04268=1024.246,392.203,-149.494,172.992,48.978,159.879
C04269=1024.236,391.958,-149.450,172.982,48.976,159.877
C04270=1024.227,391.711,-149.407,172.972,48.975,159.876
C04271=1024.218,391.466,-149.365,172.962,48.973,159.874
C04272=1024.208,391.220,-149.321,172.952,48.972,159.872
C04273=1024.199,390.973,-149.278,172.942,48.971,159.870
C04274=1024.189,390.727,-149.235,172.931,48.970,159.868
C04275=1024.180,390.481,-149.192,172.922,48.969,159.866
C04276=1024.170,390.235,-149.150,172.912,48.968,159.865
C04277=1024.162,389.990,-149.106,172.901,48.966,159.863
C04278=1024.152,389.743,-149.064,172.892,48.965,159.861
C04279=1024.142,389.498,-149.021,172.882,48.964,159.859
C04280=1024.133,389.251,-148.978,172.872,48.963,159.857
C04281=1024.124,389.005,-148.935,172.863,48.961,159.855
C04282=1024.115,388.759,-148.893,172.853,48.960,159.854
C04283=1024.105,388.513,-148.850,172.843,48.959,159.852
C04284=1024.096,388.266,-148.808,172.833,48.958,159.850
C04285=1024.087,388.020,-148.765,172.823,48.957,159.848
C04286=1024.078,387.774,-148.722,172.814,48.956,159.847
C04287=1024.069,387.528,-148.680,172.804,48.955,159.845
C04288=1024.060,387.282,-148.638,172.795,48.953,159.843
C04289=1024.050,387.035,-148.596,172.785,48.953,159.841
C04290=1024.040,386.790,-148.553,172.776,48.952,159.840
C04291=1024.032,386.543,-148.511,172.766,48.951,159.838
C04292=1024.023,386.297,-148.468,172.756,48.949,159.836
C04293=1024.014,386.050,-148.426,172.746,48.948,159.834
C04294=1024.004,385.804,-148.384,172.738,48.948,159.833
C04295=1023.995,385.558,-148.342,172.727,48.947,159.831
C04296=1023.986,385.312,-148.300,172.719,48.946,159.829
C04297=1023.977,385.066,-148.258,172.708,48.945,159.828
C04298=1023.967,384.819,-148.217,172.700,48.944,159.826
C04299=1023.958,384.573,-148.175,172.690,48.943,159.824
C04300=1023.949,384.327,-148.132,172.681,48.942,159.823
C04301=1023.940,384.081,-148.091,172.671,48.941,159.821
C04302=1023.931,383.834,-148.049,172.662,48.941,159.819
C04303=1023.922,383.588,-148.007,172.653,48.939,159.818
C04304=1023.913,383.342,-147.965,172.643,48.939,159.816
C04305=1023.904,383.095,-147.924,172.634,48.938,159.815
C04306=1023.894,382.849,-147.883,172.624,48.937,159.813
C04307=1023.885,382.603,-147.841,172.615,48.936,159.811
C04308=1023.877,382.357,-147.799,172.606,48.936,159.810
C04309=1023.868,382.110,-147.758,172.597,48.935,159.808
C04310=1023.859,381.864,-147.716,172.588,48.935,159.807
C04311=1023.850,381.617,-147.674,172.579,48.933,159.805
C04312=1023.841,381.371,-147.632,172.569,48.933,159.803
C04313=1023.832,381.119,-147.590,172.560,48.932,159.802
C04314=1023.822,380.869,-147.548,172.550,48.932,159.800
C04315=1023.814,380.618,-147.506,172.541,48.931,159.799
C04316=1023.805,380.366,-147.464,172.533,48.930,159.797
C04317=1023.796,380.119,-147.422,172.523,48.930,159.795
C04318=1023.787,379.873,-147.380,172.514,48.929,159.794
C04319=1023.779,379.627,-147.340,172.505,48.928,159.792
C04320=1023.770,379.380,-147.298,172.496,48.927,159.791
C04321=1023.760,379.134,-147.257,172.488,48.927,159.789
C04322=1023.752,378.887,-147.216,172.478,48.926,159.788
C04323=1023.743,378.642,-147.174,172.469,48.925,159.786
C04324=1023.735,378.395,-147.133,172.460,48.925,159.785
C04325=1023.726,378.148,-147.092,172.452,48.924,159.783
C04326=1023.718,377.902,-147.051,172.443,48.924,159.782
C04327=1023.709,377.656,-147.009,172.434,48.923,159.780
C04328=1023.700,377.409,-146.968,172.425,48.922,159.779
C04329=1023.691,377.163,-146.928,172.416,48.922,159.777
C04330=1023.682,376.916,-146.887,172.407,48.921,159.776
C04331=1023.674,376.670,-146.846,172.398,48.921,159.774
C04332=1023.666,376.423,-146.805,172.390,48.921,159.773
C04333=1023.656,376.176,-146.765,172.381,48.920,159.772
C04334=1023.648,375.930,-146.724,172.373,48.920,159.770
C04335=1023.639,375.684,-146.683,172.364,48.919,159.769
C04336=1023.631,375.438,-146.642,172.355,48.919,159.767
C04337=1023.621,375.191,-146.602,172.346,48.919,159.766
C04338=1023.613,374.945,-146.561,172.337,48.918,159.764
C04339=1023.605,374.697,-146.521,172.329,48.918,159.763
C04340=1023.596,374.451,-146.481,172.321,48.918,159.762
C04341=1023.587,374.204,-146.440,172.312,48.917,159.760
C04342=1023.579,373.958,-146.400,172.303,48.917,159.759
C04343=1023.570,373.711,-146.359,172.295,48.916,159.758
C04344=1023.561,373.465,-146.319,172.286,48.916,159.756
C04345=1023.553,373.219,-146.278,172.278,48.916,159.755
C04346=1023.544,372.972,-146.238,172.269,48.915,159.753
C04347=1023.536,372.726,-146.198,172.261,48.915,159.752
C04348=1023.527,372.479,-146.157,172.252,48.915,159.751
C04349=1023.519,372.232,-146.117,172.244,48.915,159.749
C04350=1023.510,371.986,-146.077,172.235,48.915,159.748
C04351=1023.502,371.739,-146.036,172.227,48.914,159.747
C04352=1023.493,371.492,-145.997,172.219,48.914,159.745
C04353=1023.485,371.246,-145.956,172.210,48.914,159.744
C04354=1023.477,371.000,-145.917,172.202,48.914,159.743
C04355=1023.468,370.753,-145.876,172.194,48.913,159.742
C04356=1023.460,370.506,-145.836,172.186,48.913,159.740
C04357=1023.452,370.260,-145.796,172.177,48.913,159.739
C04358=1023.444,370.013,-145.756,172.169,48.913,159.738
C04359=1023.435,369.767,-145.716,172.161,48.913,159.736
C04360=1023.427,369.519,-145.676,172.152,48.912,159.735
C04361=1023.418,369.273,-145.637,172.144,48.912,159.734
C04362=1023.410,369.026,-145.596,172.136,48.913,159.733
C04363=1023.402,368.780,-145.557,172.128,48.912,159.731
C04364=1023.394,368.533,-145.517,172.120,48.912,159.730
C04365=1023.386,368.286,-145.477,172.111,48.912,159.729
C04366=1023.377,368.040,-145.438,172.103,48.912,159.728
C04367=1023.370,367.793,-145.398,172.095,48.912,159.726
C04368=1023.361,367.545,-145.358,172.087,48.912,159.725
C04369=1023.353,367.308,-145.320,172.079,48.912,159.724
C04370=1023.344,367.070,-145.283,172.071,48.912,159.723
C04371=1023.336,366.832,-145.245,172.064,48.912,159.721
C04372=1023.328,366.594,-145.206,172.056,48.912,159.720
C04373=1023.320,366.355,-145.168,172.048,48.912,159.719
C04374=1023.312,366.117,-145.130,172.040,48.912,159.718
C04375=1023.305,365.879,-145.092,172.032,48.912,159.717
C04376=1023.297,365.641,-145.055,172.025,48.912,159.716
C04377=1023.288,365.394,-145.015,172.017,48.912,159.714
C04378=1023.280,365.148,-144.976,172.008,48.913,159.713
C04379=1023.272,364.901,-144.937,172.001,48.913,159.712
C04380=1023.263,364.654,-144.898,171.993,48.913,159.711
C04381=1023.256,364.407,-144.858,171.985,48.913,159.710
C04382=1023.247,364.160,-144.819,171.977,48.913,159.709
C04383=1023.239,363.913,-144.780,171.970,48.913,159.708
C04384=1023.231,363.667,-144.741,171.961,48.913,159.706
C04385=1023.223,363.421,-144.702,171.953,48.914,159.705
C04386=1023.215,363.174,-144.663,171.946,48.914,159.704
C04387=1023.207,362.927,-144.623,171.938,48.914,159.703
C04388=1023.199,362.679,-144.585,171.930,48.914,159.702
C04389=1023.190,362.433,-144.545,171.923,48.915,159.701
C04390=1023.183,362.186,-144.507,171.915,48.915,159.700
C04391=1023.174,361.940,-144.468,171.906,48.915,159.698
C04392=1023.167,361.692,-144.429,171.899,48.915,159.697
C04393=1023.159,361.445,-144.390,171.891,48.915,159.696
C04394=1023.151,361.199,-144.351,171.883,48.916,159.695
C04395=1023.143,360.952,-144.312,171.876,48.916,159.694
C04396=1023.134,360.705,-144.273,171.868,48.916,159.693
C04397=1023.127,360.459,-144.235,171.861,48.916,159.692
C04398=1023.119,360.211,-144.196,171.853,48.917,159.691
C04399=1023.111,359.964,-144.157,171.845,48.918,159.690
C04400=1023.104,359.718,-144.119,171.838,48.918,159.689
C04401=1023.095,359.470,-144.080,171.830,48.918,159.688
C04402=1023.086,359.224,-144.041,171.823,48.918,159.687
C04403=1023.079,358.978,-144.003,171.815,48.919,159.686
C04404=1023.070,358.730,-143.965,171.807,48.919,159.685
C04405=1023.063,358.484,-143.926,171.800,48.920,159.684
C04406=1023.055,358.237,-143.888,171.792,48.920,159.682
C04407=1023.047,357.989,-143.849,171.785,48.921,159.682
C04408=1023.039,357.742,-143.812,171.777,48.921,159.680
C04409=1023.031,357.495,-143.773,171.770,48.921,159.679
C04410=1023.024,357.248,-143.735,171.762,48.922,159.678
C04411=1023.015,357.002,-143.697,171.754,48.922,159.677
C04412=1023.007,356.755,-143.659,171.747,48.923,159.676
C04413=1022.999,356.508,-143.620,171.739,48.924,159.675
C04414=1022.992,356.261,-143.582,171.733,48.924,159.674
C04415=1022.984,356.014,-143.544,171.725,48.925,159.673
C04416=1022.976,355.767,-143.506,171.718,48.925,159.673
C04417=1022.968,355.519,-143.468,171.710,48.926,159.671
C04418=1022.960,355.273,-143.430,171.703,48.926,159.671
C04419=1022.952,355.026,-143.392,171.695,48.927,159.669
C04420=1022.945,354.779,-143.354,171.688,48.927,159.669
C04421=1022.937,354.532,-143.316,171.680,48.928,159.668
C04422=1022.930,354.285,-143.278,171.673,48.928,159.667
C04423=1022.921,354.038,-143.240,171.666,48.929,159.666
C04424=1022.914,353.791,-143.203,171.659,48.930,159.665
C04425=1022.906,353.544,-143.164,171.652,48.931,159.664
C04426=1022.898,353.297,-143.127,171.644,48.931,159.663
C04427=1022.890,353.050,-143.090,171.637,48.932,159.662
C04428=1022.882,352.803,-143.051,171.630,48.933,159.661
C04429=1022.875,352.568,-143.016,171.623,48.934,159.660
C04430=1022.867,352.333,-142.980,171.616,48.934,159.659
C04431=1022.860,352.099,-142.944,171.609,48.935,159.658
C04432=1022.852,351.864,-142.909,171.603,48.936,159.658
C04433=1022.845,351.630,-142.873,171.596,48.936,159.657
C04434=1022.838,351.395,-142.837,171.589,48.937,159.656
C04435=1022.831,351.160,-142.801,171.582,48.938,159.655
C04436=1022.823,350.925,-142.766,171.575,48.939,159.654
C04437=1022.816,350.678,-142.728,171.568,48.939,159.653
C04438=1022.808,350.431,-142.691,171.561,48.940,159.652
C04439=1022.801,350.185,-142.653,171.554,48.941,159.652
C04440=1022.793,349.938,-142.616,171.547,48.942,159.651
C04441=1022.785,349.690,-142.578,171.539,48.943,159.650
C04442=1022.778,349.443,-142.541,171.532,48.943,159.649
C04443=1022.770,349.196,-142.504,171.526,48.944,159.648
C04444=1022.762,348.949,-142.466,171.518,48.945,159.647
C04445=1022.755,348.702,-142.429,171.512,48.946,159.646
C04446=1022.747,348.455,-142.392,171.505,48.947,159.646
C04447=1022.740,348.208,-142.354,171.497,48.948,159.645
C04448=1022.732,347.960,-142.318,171.490,48.949,159.644
C04449=1022.725,347.713,-142.281,171.484,48.949,159.643
C04450=1022.717,347.466,-142.244,171.476,48.951,159.642
C04451=1022.710,347.219,-142.206,171.470,48.951,159.641
C04452=1022.702,346.972,-142.169,171.463,48.952,159.641
C04453=1022.695,346.725,-142.132,171.455,48.954,159.640
C04454=1022.687,346.478,-142.095,171.449,48.954,159.639
C04455=1022.679,346.231,-142.058,171.442,48.955,159.638
C04456=1022.672,345.983,-142.022,171.435,48.957,159.637
C04457=1022.664,345.736,-141.985,171.428,48.957,159.637
C04458=1022.656,345.489,-141.948,171.421,48.959,159.636
C04459=1022.649,345.242,-141.911,171.415,48.959,159.635
C04460=1022.641,344.994,-141.875,171.407,48.960,159.634
C04461=1022.634,344.747,-141.837,171.401,48.962,159.633
C04462=1022.626,344.500,-141.800,171.394,48.962,159.633
C04463=1022.618,344.253,-141.764,171.386,48.964,159.632
C04464=1022.612,344.005,-141.727,171.380,48.965,159.631
C04465=1022.604,343.758,-141.690,171.373,48.966,159.630
C04466=1022.596,343.511,-141.654,171.367,48.967,159.630
C04467=1022.589,343.265,-141.617,171.359,48.968,159.629
C04468=1022.582,343.017,-141.581,171.353,48.969,159.628
C04469=1022.574,342.770,-141.545,171.346,48.971,159.627
C04470=1022.567,342.523,-141.507,171.340,48.971,159.627
C04471=1022.559,342.275,-141.471,171.332,48.973,159.626
C04472=1022.551,342.028,-141.435,171.326,48.974,159.625
C04473=1022.545,341.781,-141.398,171.319,48.975,159.624
C04474=1022.537,341.534,-141.361,171.313,48.976,159.624
C04475=1022.529,341.286,-141.325,171.306,48.978,159.623
C04476=1022.522,341.039,-141.289,171.299,48.979,159.622
C04477=1022.515,340.792,-141.252,171.292,48.980,159.621
C04478=1022.508,340.544,-141.216,171.286,48.981,159.621
C04479=1022.500,340.297,-141.180,171.280,48.982,159.620
C04480=1022.494,340.050,-141.143,171.273,48.984,159.619
C04481=1022.486,339.802,-141.107,171.266,48.985,159.619
C04482=1022.478,339.556,-141.070,171.259,48.987,159.618
C04483=1022.471,339.308,-141.035,171.253,48.988,159.617
C04484=1022.463,339.061,-140.999,171.247,48.989,159.617
C04485=1022.456,338.813,-140.963,171.240,48.990,159.616
C04486=1022.449,338.567,-140.927,171.233,48.992,159.615
C04487=1022.441,338.319,-140.891,171.227,48.993,159.615
C04488=1022.433,338.072,-140.854,171.220,48.995,159.614
C04489=1022.427,337.835,-140.820,171.214,48.996,159.613
C04490=1022.420,337.599,-140.785,171.207,48.997,159.613
C04491=1022.413,337.363,-140.752,171.201,48.998,159.612
C04492=1022.406,337.127,-140.717,171.196,48.999,159.611
C04493=1022.399,336.891,-140.683,171.190,49.001,159.611
C04494=1022.392,336.655,-140.649,171.183,49.003,159.610
C04495=1022.385,336.418,-140.614,171.177,49.004,159.610
C04496=1022.378,336.181,-140.580,171.170,49.005,159.609
C04497=1022.371,335.935,-140.544,171.164,49.006,159.608
C04498=1022.363,335.687,-140.508,171.158,49.008,159.608
C04499=1022.357,335.440,-140.473,171.152,49.010,159.607
C04500=1022.349,335.192,-140.437,171.145,49.011,159.607
C04501=1022.342,334.945,-140.402,171.138,49.013,159.606
C04502=1022.334,334.698,-140.366,171.132,49.014,159.605
C04503=1022.327,334.451,-140.330,171.126,49.016,159.605
C04504=1022.320,334.203,-140.294,171.119,49.017,159.604
C04505=1022.313,333.956,-140.258,171.113,49.018,159.603
C04506=1022.306,333.709,-140.223,171.107,49.020,159.603
C04507=1022.299,333.461,-140.188,171.100,49.022,159.602
C04508=1022.292,333.214,-140.152,171.094,49.023,159.602
C04509=1022.284,332.966,-140.116,171.088,49.025,159.601
C04510=1022.277,332.719,-140.081,171.082,49.026,159.600
C04511=1022.270,332.472,-140.046,171.076,49.028,159.600
C04512=1022.262,332.224,-140.010,171.068,49.030,159.599
C04513=1022.256,331.977,-139.975,171.062,49.031,159.599
C04514=1022.248,331.730,-139.940,171.056,49.033,159.598
C04515=1022.240,331.482,-139.905,171.050,49.035,159.598
C04516=1022.234,331.235,-139.869,171.044,49.037,159.597
C04517=1022.227,330.987,-139.834,171.037,49.038,159.597
C04518=1022.220,330.739,-139.799,171.031,49.040,159.596
C04519=1022.212,330.492,-139.764,171.025,49.041,159.595
C04520=1022.205,330.245,-139.729,171.019,49.043,159.595
C04521=1022.198,329.997,-139.693,171.013,49.045,159.594
C04522=1022.191,329.750,-139.658,171.006,49.046,159.594
C04523=1022.183,329.503,-139.623,171.000,49.048,159.593
C04524=1022.177,329.256,-139.588,170.994,49.050,159.593
C04525=1022.169,329.008,-139.553,170.988,49.052,159.592
C04526=1022.162,328.760,-139.517,170.982,49.053,159.592
C04527=1022.155,328.513,-139.483,170.975,49.055,159.591
C04528=1022.148,328.266,-139.448,170.969,49.057,159.591
C04529=1022.141,328.018,-139.413,170.963,49.059,159.590
C04530=1022.135,327.771,-139.378,170.956,49.061,159.590
C04531=1022.127,327.523,-139.343,170.950,49.062,159.589
C04532=1022.120,327.275,-139.308,170.944,49.064,159.589
C04533=1022.113,327.028,-139.273,170.938,49.066,159.588
C04534=1022.106,326.781,-139.239,170.932,49.068,159.588
C04535=1022.099,326.534,-139.203,170.926,49.070,159.587
C04536=1022.092,326.286,-139.170,170.920,49.072,159.587
C04537=1022.084,326.039,-139.135,170.914,49.074,159.586
C04538=1022.077,325.790,-139.100,170.908,49.076,159.586
C04539=1022.070,325.543,-139.066,170.902,49.078,159.585
C04540=1022.062,325.296,-139.031,170.896,49.080,159.585
C04541=1022.056,325.048,-138.997,170.890,49.082,159.584
C04542=1022.048,324.801,-138.962,170.884,49.083,159.584
C04543=1022.041,324.553,-138.928,170.878,49.085,159.584
C04544=1022.034,324.306,-138.893,170.872,49.087,159.583
C04545=1022.027,324.058,-138.859,170.866,49.090,159.583
C04546=1022.020,323.811,-138.825,170.860,49.092,159.582
C04547=1022.012,323.564,-138.791,170.854,49.094,159.582
C04548=1022.006,323.316,-138.757,170.848,49.096,159.581
C04549=1021.999,323.078,-138.723,170.842,49.098,159.581
C04550=1021.992,322.839,-138.690,170.837,49.100,159.581
C04551=1021.985,322.601,-138.657,170.831,49.102,159.580
C04552=1021.978,322.362,-138.624,170.825,49.104,159.580
C04553=1021.971,322.124,-138.591,170.819,49.106,159.579
C04554=1021.964,321.885,-138.558,170.814,49.108,159.579
C04555=1021.958,321.646,-138.525,170.808,49.110,159.579
C04556=1021.951,321.408,-138.492,170.803,49.112,159.578
C04557=1021.944,321.161,-138.459,170.797,49.114,159.578
C04558=1021.937,320.913,-138.425,170.791,49.116,159.577
C04559=1021.930,320.666,-138.390,170.785,49.118,159.577
C04560=1021.923,320.418,-138.356,170.779,49.121,159.577
C04561=1021.916,320.170,-138.322,170.773,49.122,159.576
C04562=1021.909,319.922,-138.288,170.767,49.124,159.576
C04563=1021.902,319.675,-138.254,170.762,49.127,159.575
C04564=1021.895,319.428,-138.219,170.756,49.129,159.575
C04565=1021.888,319.181,-138.186,170.750,49.131,159.575
C04566=1021.882,318.933,-138.151,170.744,49.133,159.574
C04567=1021.874,318.685,-138.118,170.738,49.135,159.574
C04568=1021.867,318.437,-138.084,170.732,49.138,159.574
C04569=1021.861,318.189,-138.049,170.726,49.140,159.573
C04570=1021.854,317.942,-138.016,170.720,49.142,159.573
C04571=1021.847,317.695,-137.982,170.714,49.144,159.572
C04572=1021.840,317.447,-137.948,170.709,49.147,159.572
C04573=1021.833,317.199,-137.914,170.703,49.149,159.572
C04574=1021.827,316.952,-137.880,170.698,49.151,159.571
C04575=1021.819,316.704,-137.846,170.692,49.153,159.571
C04576=1021.812,316.457,-137.813,170.686,49.155,159.571
C04577=1021.806,316.209,-137.779,170.681,49.158,159.570
C04578=1021.799,315.962,-137.745,170.675,49.160,159.570
C04579=1021.792,315.714,-137.711,170.669,49.162,159.570
C04580=1021.786,315.466,-137.678,170.663,49.165,159.569
C04581=1021.779,315.218,-137.644,170.657,49.167,159.569
C04582=1021.772,314.971,-137.610,170.651,49.169,159.569
C04583=1021.765,314.724,-137.577,170.647,49.172,159.568
C04584=1021.759,314.476,-137.542,170.641,49.174,159.568
C04585=1021.752,314.229,-137.509,170.635,49.176,159.568
C04586=1021.745,313.981,-137.476,170.629,49.179,159.567
C04587=1021.738,313.733,-137.442,170.624,49.181,159.567
C04588=1021.732,313.486,-137.408,170.618,49.183,159.567
C04589=1021.725,313.238,-137.374,170.612,49.186,159.566
C04590=1021.719,312.990,-137.341,170.606,49.188,159.566
C04591=1021.712,312.743,-137.307,170.602,49.191,159.566
C04592=1021.706,312.495,-137.273,170.596,49.193,159.565
C04593=1021.699,312.247,-137.240,170.590,49.195,159.565
C04594=1021.692,312.000,-137.207,170.584,49.198,159.565
C04595=1021.685,311.752,-137.173,170.579,49.200,159.564
C04596=1021.680,311.505,-137.139,170.573,49.203,159.564
C04597=1021.672,311.257,-137.106,170.568,49.205,159.564
C04598=1021.666,311.009,-137.073,170.563,49.208,159.564
C04599=1021.659,310.762,-137.039,170.557,49.210,159.563
C04600=1021.653,310.514,-137.006,170.551,49.212,159.563
C04601=1021.647,310.267,-136.972,170.545,49.215,159.563
C04602=1021.640,310.018,-136.939,170.539,49.217,159.562
C04603=1021.633,309.772,-136.906,170.535,49.220,159.562
C04604=1021.626,309.524,-136.873,170.529,49.223,159.562
C04605=1021.619,309.276,-136.840,170.524,49.225,159.562
C04606=1021.612,309.028,-136.808,170.518,49.228,159.562
C04607=1021.605,308.781,-136.775,170.512,49.230,159.561
C04608=1021.597,308.533,-136.742,170.507,49.233,159.561
C04609=1021.592,308.297,-136.711,170.501,49.236,159.561
C04610=1021.585,308.061,-136.680,170.497,49.238,159.561
C04611=1021.579,307.826,-136.648,170.491,49.241,159.560
C04612=1021.572,307.589,-136.617,170.485,49.243,159.560
C04613=1021.565,307.353,-136.587,170.481,49.246,159.560
C04614=1021.559,307.117,-136.555,170.475,49.249,159.560
C04615=1021.553,306.882,-136.524,170.471,49.251,159.560
C04616=1021.546,306.646,-136.493,170.465,49.254,159.559
C04617=1021.539,306.398,-136.460,170.460,49.257,159.559
C04618=1021.532,306.151,-136.428,170.454,49.259,159.559
C04619=1021.526,305.903,-136.395,170.448,49.262,159.559
C04620=1021.518,305.655,-136.362,170.444,49.265,159.559
C04621=1021.512,305.407,-136.330,170.438,49.267,159.558
C04622=1021.506,305.160,-136.297,170.433,49.271,159.558
C04623=1021.498,304.912,-136.264,170.427,49.273,159.558
C04624=1021.492,304.664,-136.232,170.422,49.276,159.558
C04625=1021.486,304.417,-136.199,170.416,49.279,159.558
C04626=1021.478,304.168,-136.167,170.411,49.282,159.557
C04627=1021.472,303.920,-136.134,170.406,49.284,159.557
C04628=1021.465,303.673,-136.102,170.401,49.287,159.557
C04629=1021.459,303.426,-136.069,170.395,49.290,159.557
C04630=1021.452,303.177,-136.036,170.390,49.293,159.557
C04631=1021.445,302.930,-136.004,170.384,49.296,159.557
C04632=1021.439,302.682,-135.972,170.379,49.299,159.556
C04633=1021.432,302.434,-135.940,170.373,49.302,159.556
C04634=1021.425,302.187,-135.907,170.369,49.305,159.556
C04635=1021.418,301.939,-135.874,170.363,49.307,159.556
C04636=1021.412,301.691,-135.843,170.358,49.310,159.556
C04637=1021.405,301.443,-135.810,170.352,49.313,159.556
C04638=1021.398,301.196,-135.778,170.347,49.316,159.555
C04639=1021.392,300.948,-135.746,170.343,49.319,159.555
C04640=1021.386,300.700,-135.713,170.337,49.322,159.555
C04641=1021.379,300.453,-135.681,170.332,49.325,159.555
C04642=1021.373,300.204,-135.649,170.326,49.328,159.555
C04643=1021.365,299.957,-135.616,170.321,49.331,159.555
C04644=1021.359,299.709,-135.584,170.315,49.334,159.555
C04645=1021.353,299.461,-135.552,170.311,49.336,159.554
C04646=1021.346,299.213,-135.520,170.305,49.339,159.554
C04647=1021.340,298.965,-135.487,170.300,49.343,159.554
C04648=1021.333,298.718,-135.455,170.295,49.346,159.554
C04649=1021.327,298.470,-135.423,170.290,49.348,159.554
C04650=1021.321,298.222,-135.391,170.285,49.351,159.554
C04651=1021.314,297.974,-135.359,170.279,49.355,159.554
C04652=1021.308,297.727,-135.326,170.274,49.358,159.554
C04653=1021.301,297.479,-135.295,170.268,49.360,159.553
C04654=1021.295,297.231,-135.262,170.264,49.363,159.553
C04655=1021.288,296.983,-135.231,170.259,49.366,159.553
C04656=1021.282,296.735,-135.199,170.254,49.370,159.553
C04657=1021.276,296.487,-135.166,170.248,49.373,159.553
C04658=1021.269,296.240,-135.135,170.244,49.376,159.553
C04659=1021.263,295.992,-135.102,170.238,49.378,159.553
C04660=1021.256,295.744,-135.070,170.233,49.382,159.553
C04661=1021.250,295.496,-135.038,170.228,49.385,159.553
C04662=1021.244,295.248,-135.006,170.223,49.388,159.553
C04663=1021.237,295.000,-134.974,170.218,49.391,159.552
C04664=1021.231,294.752,-134.942,170.213,49.394,159.552
C04665=1021.224,294.504,-134.911,170.207,49.397,159.552
C04666=1021.218,294.257,-134.878,170.203,49.400,159.552
C04667=1021.212,294.009,-134.847,170.198,49.404,159.552
C04668=1021.206,293.761,-134.815,170.192,49.407,159.552
C04669=1021.200,293.534,-134.786,170.188,49.410,159.552
C04670=1021.195,293.306,-134.756,170.182,49.412,159.552
C04671=1021.188,293.079,-134.728,170.178,49.415,159.552
C04672=1021.182,292.852,-134.698,170.174,49.418,159.552
C04673=1021.176,292.625,-134.670,170.169,49.421,159.552
C04674=1021.171,292.398,-134.641,170.164,49.424,159.552
C04675=1021.164,292.171,-134.612,170.160,49.427,159.552
C04676=1021.159,291.944,-134.583,170.155,49.430,159.552
C04677=1021.152,291.696,-134.551,170.150,49.433,159.551
C04678=1021.145,291.448,-134.520,170.145,49.437,159.552
C04679=1021.139,291.201,-134.489,170.140,49.440,159.551
C04680=1021.132,290.953,-134.458,170.135,49.444,159.551
C04681=1021.126,290.705,-134.426,170.130,49.447,159.551
C04682=1021.119,290.457,-134.395,170.125,49.450,159.551
C04683=1021.113,290.209,-134.363,170.120,49.454,159.551
C04684=1021.107,289.960,-134.332,170.115,49.457,159.551
C04685=1021.100,289.713,-134.301,170.110,49.461,159.551
C04686=1021.094,289.465,-134.269,170.105,49.464,159.551
C04687=1021.087,289.217,-134.238,170.100,49.467,159.551
C04688=1021.080,288.969,-134.207,170.095,49.471,159.551
C04689=1021.074,288.721,-134.176,170.090,49.474,159.551
C04690=1021.068,288.474,-134.145,170.084,49.477,159.551
C04691=1021.061,288.226,-134.113,170.080,49.481,159.551
C04692=1021.055,287.977,-134.083,170.075,49.484,159.551
C04693=1021.049,287.729,-134.051,170.070,49.488,159.551
C04694=1021.043,287.482,-134.020,170.065,49.491,159.551
C04695=1021.036,287.233,-133.989,170.061,49.495,159.551
C04696=1021.029,286.985,-133.957,170.056,49.498,159.551
C04697=1021.023,286.738,-133.926,170.051,49.502,159.551
C04698=1021.017,286.490,-133.896,170.045,49.505,159.551
C04699=1021.010,286.242,-133.864,170.040,49.509,159.551
C04700=1021.004,285.994,-133.834,170.036,49.512,159.551
C04701=1020.998,285.746,-133.802,170.031,49.516,159.551
C04702=1020.991,285.497,-133.772,170.026,49.519,159.551
C04703=1020.984,285.250,-133.740,170.021,49.523,159.551
C04704=1020.979,285.002,-133.710,170.017,49.526,159.551
C04705=1020.971,284.754,-133.679,170.012,49.530,159.551
C04706=1020.965,284.506,-133.648,170.007,49.534,159.552
C04707=1020.959,284.258,-133.618,170.001,49.537,159.551
C04708=1020.952,284.010,-133.587,169.996,49.541,159.552
C04709=1020.946,283.761,-133.556,169.991,49.545,159.552
C04710=1020.939,283.514,-133.526,169.987,49.548,159.552
C04711=1020.932,283.266,-133.495,169.982,49.551,159.552
C04712=1020.927,283.018,-133.464,169.977,49.555,159.552
C04713=1020.920,282.770,-133.434,169.972,49.559,159.552
C04714=1020.914,282.522,-133.402,169.967,49.563,159.552
C04715=1020.907,282.274,-133.372,169.963,49.566,159.552
C04716=1020.901,282.026,-133.342,169.958,49.570,159.552
C04717=1020.895,281.778,-133.311,169.953,49.574,159.552
C04718=1020.888,281.529,-133.281,169.948,49.578,159.552
C04719=1020.882,281.281,-133.249,169.943,49.582,159.552
C04720=1020.875,281.034,-133.219,169.939,49.585,159.552
C04721=1020.869,280.785,-133.189,169.934,49.589,159.552
C04722=1020.863,280.538,-133.158,169.929,49.592,159.553
C04723=1020.856,280.289,-133.128,169.924,49.596,159.553
C04724=1020.851,280.041,-133.097,169.920,49.600,159.553
C04725=1020.843,279.794,-133.066,169.915,49.604,159.553
C04726=1020.837,279.546,-133.036,169.910,49.608,159.553
C04727=1020.831,279.297,-133.005,169.905,49.611,159.553
C04728=1020.825,279.049,-132.975,169.900,49.615,159.553
C04729=1020.819,278.828,-132.949,169.896,49.618,159.553
C04730=1020.814,278.608,-132.921,169.892,49.622,159.553
C04731=1020.808,278.386,-132.894,169.888,49.625,159.553
C04732=1020.803,278.166,-132.867,169.884,49.629,159.553
C04733=1020.797,277.944,-132.840,169.880,49.632,159.554
C04734=1020.791,277.723,-132.813,169.876,49.635,159.554
C04735=1020.786,277.503,-132.786,169.871,49.639,159.554
C04736=1020.780,277.281,-132.759,169.867,49.643,159.554
C04737=1020.774,277.033,-132.728,169.863,49.646,159.554
C04738=1020.767,276.785,-132.698,169.858,49.650,159.554
C04739=1020.761,276.537,-132.668,169.853,49.654,159.554
C04740=1020.755,276.290,-132.638,169.848,49.658,159.554
C04741=1020.748,276.041,-132.607,169.843,49.662,159.554
C04742=1020.742,275.793,-132.578,169.839,49.665,159.555
C04743=1020.736,275.544,-132.547,169.834,49.669,159.555
C04744=1020.730,275.297,-132.517,169.829,49.673,159.555
C04745=1020.723,275.049,-132.487,169.824,49.678,159.555
C04746=1020.717,274.801,-132.457,169.820,49.682,159.555
C04747=1020.711,274.552,-132.428,169.816,49.685,159.555
C04748=1020.705,274.305,-132.397,169.811,49.689,159.555
C04749=1020.698,274.056,-132.367,169.806,49.693,159.555
C04750=1020.692,273.808,-132.337,169.801,49.698,159.556
C04751=1020.686,273.560,-132.308,169.796,49.702,159.556
C04752=1020.679,273.312,-132.277,169.792,49.705,159.556
C04753=1020.673,273.064,-132.248,169.788,49.710,159.556
C04754=1020.667,272.816,-132.218,169.783,49.714,159.556
C04755=1020.660,272.568,-132.188,169.778,49.718,159.556
C04756=1020.654,272.319,-132.158,169.773,49.722,159.557
C04757=1020.648,272.072,-132.128,169.769,49.726,159.557
C04758=1020.642,271.823,-132.098,169.764,49.730,159.557
C04759=1020.635,271.575,-132.068,169.760,49.734,159.557
C04760=1020.629,271.327,-132.039,169.755,49.738,159.557
C04761=1020.623,271.079,-132.009,169.750,49.742,159.557
C04762=1020.616,270.830,-131.980,169.746,49.746,159.558
C04763=1020.611,270.583,-131.949,169.741,49.750,159.558
C04764=1020.604,270.334,-131.920,169.737,49.755,159.558
C04765=1020.598,270.086,-131.889,169.732,49.759,159.558
C04766=1020.592,269.838,-131.860,169.727,49.763,159.558
C04767=1020.585,269.590,-131.831,169.723,49.767,159.559
C04768=1020.580,269.342,-131.801,169.718,49.771,159.559
C04769=1020.573,269.094,-131.772,169.714,49.776,159.559
C04770=1020.566,268.845,-131.742,169.709,49.779,159.559
C04771=1020.561,268.597,-131.712,169.704,49.784,159.559
C04772=1020.554,268.349,-131.683,169.701,49.788,159.560
C04773=1020.548,268.101,-131.653,169.696,49.792,159.560
C04774=1020.541,267.853,-131.624,169.691,49.797,159.560
C04775=1020.535,267.604,-131.594,169.686,49.801,159.560
C04776=1020.529,267.357,-131.565,169.682,49.805,159.561
C04777=1020.523,267.108,-131.536,169.677,49.810,159.561
C04778=1020.516,266.860,-131.507,169.673,49.814,159.561
C04779=1020.511,266.612,-131.477,169.669,49.818,159.561
C04780=1020.504,266.363,-131.448,169.664,49.822,159.561
C04781=1020.498,266.116,-131.418,169.659,49.827,159.562
C04782=1020.491,265.867,-131.389,169.654,49.831,159.562
C04783=1020.486,265.619,-131.359,169.651,49.835,159.562
C04784=1020.479,265.371,-131.330,169.646,49.839,159.562
C04785=1020.473,265.123,-131.301,169.641,49.844,159.563
C04786=1020.467,264.875,-131.272,169.637,49.849,159.563
C04787=1020.461,264.626,-131.243,169.632,49.853,159.563
C04788=1020.454,264.378,-131.214,169.627,49.857,159.563
C04789=1020.449,264.159,-131.187,169.624,49.861,159.564
C04790=1020.444,263.941,-131.162,169.620,49.865,159.564
C04791=1020.437,263.722,-131.136,169.616,49.869,159.564
C04792=1020.432,263.504,-131.111,169.612,49.873,159.564
C04793=1020.427,263.285,-131.084,169.608,49.877,159.565
C04794=1020.421,263.065,-131.059,169.604,49.881,159.565
C04795=1020.416,262.847,-131.034,169.600,49.885,159.565
C04796=1020.410,262.629,-131.008,169.596,49.888,159.565
C04797=1020.404,262.381,-130.979,169.591,49.893,159.565
C04798=1020.399,262.132,-130.950,169.588,49.897,159.566
C04799=1020.392,261.884,-130.920,169.583,49.902,159.566
C04800=1020.385,261.635,-130.891,169.579,49.906,159.566
C04801=1020.379,261.387,-130.862,169.574,49.911,159.567
C04802=1020.373,261.139,-130.834,169.570,49.916,159.567
C04803=1020.367,260.890,-130.805,169.565,49.920,159.567
C04804=1020.361,260.642,-130.776,169.561,49.925,159.568
C04805=1020.354,260.394,-130.747,169.557,49.929,159.568
C04806=1020.348,260.146,-130.718,169.552,49.934,159.568
C04807=1020.342,259.898,-130.689,169.548,49.938,159.568
C04808=1020.337,259.650,-130.661,169.543,49.943,159.569
C04809=1020.330,259.402,-130.632,169.539,49.948,159.569
C04810=1020.323,259.153,-130.603,169.534,49.952,159.569
C04811=1020.317,258.904,-130.574,169.530,49.957,159.569
C04812=1020.310,258.657,-130.546,169.525,49.962,159.570
C04813=1020.304,258.408,-130.518,169.521,49.967,159.570
C04814=1020.298,258.160,-130.489,169.517,49.971,159.571
C04815=1020.292,257.912,-130.461,169.513,49.976,159.571
C04816=1020.285,257.664,-130.432,169.508,49.980,159.571
C04817=1020.279,257.415,-130.404,169.504,49.986,159.572
C04818=1020.272,257.167,-130.375,169.499,49.990,159.572
C04819=1020.266,256.919,-130.347,169.495,49.995,159.572
C04820=1020.260,256.670,-130.318,169.491,50.000,159.573
C04821=1020.254,256.422,-130.290,169.486,50.005,159.573
C04822=1020.247,256.174,-130.261,169.482,50.009,159.573
C04823=1020.241,255.925,-130.233,169.477,50.014,159.573
C04824=1020.234,255.677,-130.205,169.473,50.019,159.574
C04825=1020.228,255.428,-130.176,169.468,50.024,159.574
C04826=1020.222,255.180,-130.147,169.465,50.028,159.575
C04827=1020.216,254.932,-130.119,169.460,50.033,159.575
C04828=1020.209,254.684,-130.090,169.456,50.038,159.575
C04829=1020.204,254.436,-130.062,169.451,50.043,159.576
C04830=1020.197,254.187,-130.035,169.447,50.048,159.576
C04831=1020.191,253.939,-130.006,169.443,50.053,159.576
C04832=1020.185,253.690,-129.977,169.438,50.058,159.577
C04833=1020.178,253.442,-129.950,169.434,50.062,159.577
C04834=1020.172,253.194,-129.921,169.429,50.067,159.577
C04835=1020.166,252.945,-129.892,169.425,50.072,159.578
C04836=1020.160,252.697,-129.865,169.421,50.077,159.578
C04837=1020.154,252.449,-129.836,169.417,50.082,159.579
C04838=1020.148,252.200,-129.808,169.413,50.087,159.579
C04839=1020.141,251.952,-129.780,169.409,50.092,159.579
C04840=1020.135,251.703,-129.751,169.404,50.097,159.580
C04841=1020.130,251.456,-129.723,169.400,50.102,159.580
C04842=1020.123,251.207,-129.695,169.395,50.106,159.580
C04843=1020.117,250.959,-129.667,169.391,50.112,159.581
C04844=1020.111,250.710,-129.638,169.387,50.116,159.581
C04845=1020.105,250.463,-129.610,169.383,50.122,159.582
C04846=1020.099,250.214,-129.582,169.378,50.126,159.582
C04847=1020.093,249.965,-129.554,169.374,50.132,159.582
C04848=1020.086,249.717,-129.526,169.370,50.136,159.583
C04849=1020.082,249.498,-129.501,169.366,50.141,159.583
C04850=1020.076,249.278,-129.475,169.362,50.145,159.583
C04851=1020.071,249.059,-129.451,169.359,50.149,159.584
C04852=1020.065,248.839,-129.426,169.355,50.154,159.584
C04853=1020.059,248.619,-129.401,169.351,50.159,159.585
C04854=1020.054,248.400,-129.377,169.347,50.163,159.585
C04855=1020.049,248.180,-129.352,169.344,50.167,159.585
C04856=1020.043,247.961,-129.327,169.340,50.172,159.586
C04857=1020.037,247.713,-129.299,169.336,50.176,159.586
C04858=1020.031,247.464,-129.270,169.332,50.182,159.586
C04859=1020.025,247.216,-129.243,169.327,50.187,159.587
C04860=1020.019,246.967,-129.215,169.323,50.192,159.587
C04861=1020.013,246.719,-129.186,169.319,50.197,159.588
C04862=1020.007,246.471,-129.159,169.315,50.202,159.588
C04863=1020.001,246.222,-129.131,169.310,50.207,159.588
C04864=1019.996,245.974,-129.103,169.307,50.212,159.589
C04865=1019.989,245.726,-129.075,169.303,50.217,159.589
C04866=1019.983,245.477,-129.047,169.298,50.222,159.590
C04867=1019.978,245.229,-129.019,169.294,50.227,159.590
C04868=1019.971,244.980,-128.991,169.290,50.233,159.591
C04869=1019.966,244.732,-128.963,169.286,50.238,159.591
C04870=1019.959,244.484,-128.935,169.281,50.243,159.591
C04871=1019.954,244.235,-128.907,169.277,50.248,159.592
C04872=1019.948,243.987,-128.879,169.273,50.253,159.592
C04873=1019.941,243.739,-128.851,169.269,50.259,159.593
C04874=1019.936,243.490,-128.824,169.266,50.264,159.593
C04875=1019.931,243.241,-128.796,169.261,50.268,159.593
C04876=1019.924,242.994,-128.768,169.257,50.273,159.594
C04877=1019.918,242.745,-128.741,169.253,50.279,159.594
C04878=1019.912,242.496,-128.712,169.248,50.284,159.595
C04879=1019.906,242.248,-128.686,169.244,50.289,159.595
C04880=1019.899,242.000,-128.658,169.240,50.295,159.596
C04881=1019.894,241.751,-128.630,169.236,50.300,159.596
C04882=1019.888,241.502,-128.603,169.232,50.305,159.597
C04883=1019.882,241.255,-128.576,169.228,50.311,159.597
C04884=1019.876,241.006,-128.547,169.224,50.316,159.598
C04885=1019.870,240.758,-128.521,169.219,50.321,159.598
C04886=1019.863,240.509,-128.493,169.215,50.327,159.599
C04887=1019.858,240.261,-128.465,169.211,50.332,159.599
C04888=1019.851,240.012,-128.438,169.207,50.337,159.600
C04889=1019.846,239.764,-128.410,169.203,50.343,159.600
C04890=1019.839,239.516,-128.382,169.199,50.348,159.600
C04891=1019.834,239.267,-128.356,169.194,50.353,159.601
C04892=1019.827,239.019,-128.328,169.191,50.359,159.602
C04893=1019.822,238.770,-128.301,169.187,50.365,159.602
C04894=1019.815,238.522,-128.273,169.182,50.370,159.603
C04895=1019.809,238.273,-128.246,169.178,50.376,159.603
C04896=1019.803,238.025,-128.218,169.174,50.381,159.603
C04897=1019.797,237.776,-128.192,169.170,50.387,159.604
C04898=1019.791,237.527,-128.165,169.166,50.392,159.605
C04899=1019.785,237.280,-128.137,169.162,50.398,159.605
C04900=1019.778,237.031,-128.110,169.158,50.403,159.606
C04901=1019.772,236.783,-128.083,169.154,50.409,159.606
C04902=1019.766,236.534,-128.056,169.150,50.414,159.607
C04903=1019.760,236.285,-128.029,169.146,50.420,159.607
C04904=1019.755,236.037,-128.001,169.142,50.426,159.608
C04905=1019.748,235.788,-127.974,169.138,50.431,159.608
C04906=1019.742,235.540,-127.948,169.133,50.437,159.609
C04907=1019.736,235.292,-127.920,169.129,50.443,159.609
C04908=1019.730,235.043,-127.893,169.125,50.448,159.610
C04909=1019.724,234.820,-127.870,169.122,50.453,159.610
C04910=1019.719,234.598,-127.846,169.118,50.458,159.611
C04911=1019.713,234.375,-127.821,169.115,50.463,159.611
C04912=1019.707,234.152,-127.797,169.111,50.468,159.612
C04913=1019.703,233.930,-127.773,169.107,50.473,159.612
C04914=1019.697,233.707,-127.749,169.104,50.478,159.613
C04915=1019.691,233.484,-127.725,169.100,50.484,159.613
C04916=1019.686,233.261,-127.701,169.096,50.489,159.614
C04917=1019.680,233.013,-127.673,169.092,50.494,159.614
C04918=1019.674,232.764,-127.646,169.089,50.500,159.615
C04919=1019.668,232.516,-127.620,169.084,50.505,159.615
C04920=1019.662,232.267,-127.593,169.081,50.511,159.616
C04921=1019.656,232.019,-127.566,169.076,50.517,159.616
C04922=1019.650,231.770,-127.539,169.072,50.523,159.617
C04923=1019.644,231.522,-127.512,169.068,50.528,159.617
C04924=1019.638,231.273,-127.485,169.064,50.534,159.618
C04925=1019.632,231.025,-127.458,169.060,50.540,159.619
C04926=1019.626,230.776,-127.431,169.056,50.546,159.619
C04927=1019.620,230.528,-127.405,169.052,50.551,159.620
C04928=1019.614,230.279,-127.378,169.048,50.557,159.620
C04929=1019.608,230.031,-127.351,169.044,50.563,159.621
C04930=1019.602,229.782,-127.324,169.040,50.569,159.622
C04931=1019.596,229.534,-127.298,169.037,50.575,159.622
C04932=1019.590,229.285,-127.271,169.033,50.581,159.623
C04933=1019.585,229.037,-127.245,169.028,50.586,159.623
C04934=1019.578,228.788,-127.218,169.024,50.593,159.624
C04935=1019.572,228.540,-127.191,169.020,50.599,159.625
C04936=1019.566,228.291,-127.165,169.016,50.604,159.625
C04937=1019.560,228.043,-127.138,169.012,50.610,159.626
C04938=1019.554,227.794,-127.111,169.009,50.616,159.626
C04939=1019.548,227.546,-127.084,169.004,50.621,159.627
C04940=1019.542,227.297,-127.058,169.001,50.627,159.627
C04941=1019.536,227.049,-127.032,168.997,50.634,159.628
C04942=1019.529,226.800,-127.005,168.992,50.640,159.629
C04943=1019.524,226.551,-126.979,168.988,50.645,159.629
C04944=1019.518,226.303,-126.952,168.984,50.651,159.630
C04945=1019.512,226.055,-126.926,168.981,50.657,159.630
C04946=1019.506,225.806,-126.899,168.977,50.663,159.631
C04947=1019.499,225.557,-126.874,168.972,50.670,159.632
C04948=1019.493,225.309,-126.847,168.969,50.676,159.632
C04949=1019.488,225.060,-126.820,168.965,50.682,159.633
C04950=1019.481,224.812,-126.794,168.961,50.688,159.634
C04951=1019.476,224.563,-126.768,168.957,50.694,159.634
C04952=1019.468,224.314,-126.742,168.954,50.700,159.635
C04953=1019.463,224.066,-126.715,168.949,50.707,159.636
C04954=1019.457,223.817,-126.689,168.945,50.713,159.636
C04955=1019.451,223.569,-126.663,168.941,50.719,159.637
C04956=1019.445,223.321,-126.637,168.938,50.725,159.638
C04957=1019.439,223.072,-126.611,168.934,50.731,159.638
C04958=1019.432,222.823,-126.584,168.929,50.737,159.639
C04959=1019.427,222.574,-126.559,168.926,50.743,159.640
C04960=1019.420,222.326,-126.532,168.922,50.749,159.640
C04961=1019.415,222.078,-126.506,168.918,50.755,159.641
C04962=1019.408,221.829,-126.480,168.913,50.762,159.641
C04963=1019.403,221.581,-126.454,168.910,50.768,159.642
C04964=1019.397,221.332,-126.428,168.906,50.774,159.643
C04965=1019.391,221.084,-126.402,168.902,50.780,159.643
C04966=1019.385,220.835,-126.376,168.899,50.786,159.644
C04967=1019.378,220.586,-126.349,168.894,50.793,159.645
C04968=1019.372,220.337,-126.323,168.890,50.799,159.645
C04969=1019.367,220.111,-126.299,168.887,50.804,159.646
C04970=1019.362,219.884,-126.276,168.883,50.810,159.646
C04971=1019.356,219.657,-126.252,168.880,50.816,159.647
C04972=1019.351,219.430,-126.228,168.877,50.822,159.648
C04973=1019.346,219.203,-126.204,168.873,50.827,159.648
C04974=1019.340,218.977,-126.181,168.869,50.833,159.649
C04975=1019.334,218.749,-126.157,168.865,50.839,159.650
C04976=1019.329,218.523,-126.133,168.862,50.844,159.650
C04977=1019.324,218.274,-126.107,168.859,50.850,159.651
C04978=1019.317,218.026,-126.081,168.854,50.858,159.652
C04979=1019.311,217.777,-126.056,168.851,50.864,159.652
C04980=1019.305,217.529,-126.030,168.847,50.870,159.653
C04981=1019.299,217.280,-126.004,168.842,50.877,159.654
C04982=1019.293,217.031,-125.979,168.839,50.883,159.654
C04983=1019.286,216.783,-125.953,168.835,50.889,159.655
C04984=1019.281,216.534,-125.927,168.831,50.896,159.656
C04985=1019.275,216.285,-125.901,168.827,50.902,159.657
C04986=1019.269,216.037,-125.876,168.824,50.909,159.657
C04987=1019.262,215.789,-125.850,168.820,50.915,159.658
C04988=1019.257,215.540,-125.824,168.815,50.921,159.659
C04989=1019.250,215.291,-125.799,168.812,50.928,159.659
C04990=1019.244,215.042,-125.773,168.808,50.934,159.660
C04991=1019.239,214.793,-125.747,168.804,50.941,159.661
C04992=1019.232,214.545,-125.721,168.800,50.948,159.662
C04993=1019.226,214.297,-125.696,168.797,50.954,159.662
C04994=1019.220,214.048,-125.670,168.792,50.961,159.663
C04995=1019.214,213.799,-125.645,168.789,50.968,159.664
C04996=1019.208,213.550,-125.619,168.785,50.974,159.665
C04997=1019.202,213.302,-125.594,168.781,50.981,159.665
C04998=1019.196,213.053,-125.567,168.777,50.987,159.666
C04999=1019.190,212.805,-125.542,168.774,50.994,159.667
C05000=1019.184,212.556,-125.517,168.769,51.000,159.667
C05001=1019.179,212.308,-125.491,168.766,51.007,159.668
C05002=1019.173,212.059,-125.466,168.762,51.013,159.669
C05003=1019.166,211.810,-125.440,168.758,51.020,159.670
C05004=1019.160,211.562,-125.415,168.754,51.026,159.670
C05005=1019.155,211.313,-125.389,168.751,51.033,159.671
C05006=1019.149,211.064,-125.364,168.747,51.040,159.672
C05007=1019.142,210.815,-125.339,168.743,51.046,159.673
C05008=1019.137,210.566,-125.313,168.740,51.053,159.674
C05009=1019.131,210.318,-125.287,168.735,51.060,159.674
C05010=1019.125,210.070,-125.262,168.732,51.066,159.675
C05011=1019.119,209.821,-125.237,168.728,51.074,159.676
C05012=1019.113,209.572,-125.212,168.724,51.080,159.676
C05013=1019.107,209.324,-125.186,168.721,51.087,159.677
C05014=1019.101,209.075,-125.160,168.716,51.094,159.678
C05015=1019.095,208.826,-125.135,168.713,51.100,159.679
C05016=1019.089,208.578,-125.110,168.708,51.107,159.679
C05017=1019.083,208.330,-125.085,168.705,51.114,159.680
C05018=1019.077,208.081,-125.059,168.702,51.121,159.681
C05019=1019.071,207.832,-125.034,168.698,51.128,159.682
C05020=1019.065,207.583,-125.009,168.694,51.135,159.683
C05021=1019.058,207.334,-124.984,168.690,51.141,159.683
C05022=1019.053,207.086,-124.959,168.686,51.148,159.684
C05023=1019.047,206.838,-124.934,168.682,51.155,159.685
C05024=1019.040,206.589,-124.908,168.679,51.162,159.686
C05025=1019.035,206.340,-124.884,168.676,51.169,159.687
C05026=1019.029,206.092,-124.859,168.671,51.176,159.688
C05027=1019.023,205.843,-124.833,168.668,51.183,159.688
C05028=1019.016,205.594,-124.808,168.664,51.190,159.689
C05029=1019.011,205.369,-124.786,168.660,51.196,159.690
C05030=1019.006,205.143,-124.762,168.658,51.202,159.691
C05031=1019.000,204.918,-124.740,168.654,51.208,159.691
C05032=1018.995,204.692,-124.718,168.651,51.215,159.692
C05033=1018.989,204.467,-124.695,168.647,51.221,159.693
C05034=1018.984,204.241,-124.673,168.644,51.228,159.694
C05035=1018.978,204.017,-124.650,168.640,51.234,159.694
C05036=1018.973,203.791,-124.627,168.637,51.241,159.695
C05037=1018.951,202.702,-124.525,168.172,51.145,159.591
C05038=1018.947,202.484,-124.505,168.169,51.152,159.592
C05039=1018.941,202.266,-124.484,168.164,51.159,159.593
C05040=1018.937,202.048,-124.463,168.160,51.166,159.593
C05041=1018.932,201.799,-124.440,168.156,51.174,159.594
C05042=1018.927,201.551,-124.417,168.151,51.182,159.595
C05043=1018.922,201.302,-124.394,168.147,51.190,159.596
C05044=1018.917,201.052,-124.370,168.142,51.198,159.597
C05045=1018.912,200.804,-124.348,168.138,51.206,159.598
C05046=1018.907,200.555,-124.324,168.133,51.214,159.598
C05047=1018.902,200.306,-124.300,168.129,51.221,159.599
C05048=1018.897,200.057,-124.277,168.124,51.230,159.600
C05049=1018.892,199.808,-124.254,168.120,51.238,159.601
C05050=1018.887,199.559,-124.231,168.116,51.245,159.602
C05051=1018.882,199.311,-124.208,168.111,51.254,159.603
C05052=1018.877,199.062,-124.185,168.106,51.262,159.604
C05053=1018.870,198.742,-124.156,168.101,51.272,159.605
C05054=1018.864,198.423,-124.126,168.096,51.283,159.606
C05055=1018.857,198.104,-124.097,168.089,51.293,159.607
C05056=1018.850,197.784,-124.068,168.084,51.303,159.608
C05057=1018.845,197.535,-124.045,168.080,51.312,159.609
C05058=1018.840,197.287,-124.022,168.076,51.320,159.610
C05059=1018.834,197.037,-124.000,168.071,51.328,159.611
C05060=1018.829,196.788,-123.977,168.067,51.336,159.612
C05061=1018.824,196.540,-123.954,168.062,51.344,159.613
C05062=1018.818,196.291,-123.931,168.058,51.352,159.614
C05063=1018.813,196.042,-123.908,168.053,51.361,159.614
C05064=1018.809,195.793,-123.885,168.049,51.368,159.615
C05065=1018.803,195.544,-123.862,168.044,51.377,159.616
C05066=1018.798,195.295,-123.840,168.041,51.385,159.617
C05067=1018.793,195.046,-123.817,168.036,51.393,159.618
C05068=1018.788,194.798,-123.794,168.032,51.402,159.619
C05069=1018.783,194.548,-123.772,168.027,51.410,159.620
C05070=1018.778,194.300,-123.749,168.023,51.418,159.621
C05071=1018.773,194.050,-123.727,168.018,51.426,159.621
C05072=1018.767,193.801,-123.704,168.015,51.434,159.622
C05073=1018.763,193.553,-123.681,168.010,51.442,159.623
C05074=1018.757,193.303,-123.658,168.006,51.450,159.624
C05075=1018.752,193.055,-123.636,168.001,51.458,159.625
C05076=1018.747,192.805,-123.613,167.997,51.466,159.626
C05077=1018.742,192.557,-123.590,167.993,51.474,159.627
C05078=1018.737,192.308,-123.568,167.989,51.483,159.628
C05079=1018.732,192.059,-123.545,167.985,51.491,159.629
C05080=1018.727,191.810,-123.523,167.980,51.499,159.629
C05081=1018.722,191.562,-123.500,167.976,51.507,159.630
C05082=1018.717,191.313,-123.478,167.971,51.516,159.631
C05083=1018.712,191.064,-123.455,167.967,51.524,159.632
C05084=1018.707,190.815,-123.433,167.963,51.532,159.633
C05085=1018.702,190.566,-123.410,167.958,51.540,159.634
C05086=1018.697,190.317,-123.388,167.955,51.548,159.635
C05087=1018.692,190.068,-123.365,167.950,51.557,159.636
C05088=1018.687,189.819,-123.343,167.946,51.565,159.637
C05089=1018.683,189.570,-123.320,167.942,51.573,159.638
C05090=1018.677,189.321,-123.297,167.938,51.581,159.638
C05091=1018.672,189.072,-123.275,167.934,51.589,159.639
C05092=1018.666,188.823,-123.252,167.930,51.597,159.640
C05093=1018.662,188.574,-123.230,167.925,51.605,159.641
C05094=1018.658,188.325,-123.208,167.921,51.613,159.642
C05095=1018.652,188.076,-123.185,167.918,51.622,159.643
C05096=1018.648,187.827,-123.163,167.913,51.630,159.644
C05097=1018.641,187.547,-123.137,167.908,51.639,159.645
C05098=1018.637,187.266,-123.112,167.904,51.648,159.646
C05099=1018.630,186.985,-123.087,167.898,51.657,159.647
C05100=1018.625,186.704,-123.062,167.894,51.666,159.648
C05101=1018.620,186.456,-123.040,167.890,51.674,159.649
C05102=1018.615,186.206,-123.017,167.887,51.683,159.650
C05103=1018.611,185.957,-122.995,167.882,51.691,159.651
C05104=1018.606,185.709,-122.972,167.878,51.699,159.652
C05105=1018.601,185.459,-122.949,167.874,51.707,159.653
C05106=1018.596,185.210,-122.928,167.869,51.716,159.653
C05107=1018.591,184.961,-122.906,167.865,51.724,159.654
C05108=1018.585,184.712,-122.883,167.862,51.732,159.655
C05109=1018.581,184.463,-122.860,167.858,51.740,159.656
C05110=1018.577,184.214,-122.838,167.853,51.749,159.657
C05111=1018.572,183.966,-122.817,167.849,51.757,159.658
C05112=1018.567,183.716,-122.794,167.846,51.765,159.659
C05113=1018.562,183.468,-122.771,167.842,51.773,159.660
C05114=1018.557,183.219,-122.749,167.837,51.781,159.661
C05115=1018.552,182.970,-122.727,167.833,51.789,159.662
C05116=1018.548,182.720,-122.705,167.829,51.797,159.663
C05117=1018.543,182.471,-122.683,167.826,51.806,159.664
C05118=1018.538,182.223,-122.661,167.821,51.814,159.664
C05119=1018.533,181.973,-122.638,167.817,51.822,159.665
C05120=1018.528,181.724,-122.617,167.813,51.830,159.666
C05121=1018.523,181.475,-122.595,167.809,51.839,159.667
C05122=1018.518,181.227,-122.573,167.805,51.847,159.668
C05123=1018.512,180.977,-122.551,167.802,51.856,159.669
C05124=1018.507,180.729,-122.530,167.797,51.864,159.670
C05125=1018.503,180.479,-122.508,167.793,51.872,159.671
C05126=1018.497,180.231,-122.487,167.789,51.881,159.672
C05127=1018.492,179.981,-122.465,167.785,51.889,159.673
C05128=1018.487,179.732,-122.443,167.782,51.898,159.674
C05129=1018.481,179.483,-122.422,167.777,51.906,159.675
C05130=1018.477,179.234,-122.401,167.773,51.915,159.676
C05131=1018.471,178.985,-122.378,167.769,51.923,159.677
C05132=1018.466,178.736,-122.357,167.765,51.932,159.678
C05133=1018.461,178.487,-122.336,167.761,51.940,159.679
C05134=1018.456,178.238,-122.315,167.758,51.949,159.680
C05135=1018.451,177.990,-122.293,167.753,51.957,159.681
C05136=1018.446,177.739,-122.271,167.750,51.966,159.682
C05137=1018.440,177.491,-122.250,167.745,51.974,159.683
C05138=1018.435,177.242,-122.228,167.741,51.982,159.684
C05139=1018.430,176.993,-122.206,167.738,51.991,159.685
C05140=1018.425,176.744,-122.186,167.733,51.999,159.686
C05141=1018.420,176.495,-122.164,167.730,52.008,159.687
C05142=1018.415,176.245,-122.142,167.726,52.016,159.688
C05143=1018.410,175.997,-122.121,167.722,52.025,159.689
C05144=1018.405,175.748,-122.099,167.718,52.033,159.690
C05145=1018.400,175.499,-122.079,167.714,52.042,159.691
C05146=1018.395,175.250,-122.057,167.710,52.050,159.692
C05147=1018.390,175.001,-122.035,167.706,52.059,159.693
C05148=1018.385,174.752,-122.014,167.702,52.067,159.694
C05149=1018.380,174.503,-121.993,167.699,52.075,159.695
C05150=1018.375,174.253,-121.971,167.695,52.084,159.696
C05151=1018.369,174.005,-121.950,167.690,52.092,159.696
C05152=1018.365,173.755,-121.929,167.687,52.101,159.698
C05153=1018.360,173.506,-121.907,167.683,52.109,159.699
C05154=1018.354,173.258,-121.885,167.679,52.118,159.700
C05155=1018.350,173.008,-121.864,167.675,52.126,159.700
C05156=1018.344,172.760,-121.843,167.672,52.135,159.702
C05157=1018.340,172.510,-121.822,167.668,52.143,159.703
C05158=1018.335,172.262,-121.800,167.664,52.152,159.704
C05159=1018.330,172.013,-121.780,167.660,52.160,159.704
C05160=1018.325,171.764,-121.758,167.656,52.168,159.705
C05161=1018.320,171.482,-121.734,167.652,52.178,159.707
C05162=1018.314,171.200,-121.710,167.648,52.188,159.708
C05163=1018.308,170.920,-121.686,167.644,52.197,159.709
C05164=1018.303,170.638,-121.662,167.639,52.207,159.710
C05165=1018.297,170.390,-121.641,167.635,52.215,159.711
C05166=1018.293,170.141,-121.620,167.632,52.224,159.712
C05167=1018.288,169.892,-121.598,167.628,52.232,159.713
C05168=1018.283,169.643,-121.577,167.624,52.240,159.714
C05169=1018.278,169.393,-121.556,167.620,52.249,159.715
C05170=1018.273,169.145,-121.535,167.616,52.257,159.716
C05171=1018.268,168.895,-121.514,167.613,52.266,159.717
C05172=1018.263,168.646,-121.492,167.609,52.274,159.718
C05173=1018.258,168.397,-121.471,167.606,52.283,159.719
C05174=1018.254,168.148,-121.450,167.601,52.291,159.720
C05175=1018.248,167.899,-121.429,167.598,52.300,159.721
C05176=1018.244,167.650,-121.408,167.594,52.308,159.722
C05177=1018.239,167.400,-121.387,167.590,52.316,159.723
C05178=1018.233,167.152,-121.365,167.587,52.325,159.724
C05179=1018.229,166.903,-121.344,167.583,52.333,159.725
C05180=1018.224,166.653,-121.324,167.580,52.342,159.726
C05181=1018.219,166.405,-121.302,167.575,52.350,159.727
C05182=1018.214,166.155,-121.281,167.572,52.359,159.728
C05183=1018.209,165.906,-121.260,167.568,52.367,159.729
C05184=1018.205,165.658,-121.239,167.565,52.375,159.730
C05185=1018.200,165.409,-121.218,167.561,52.384,159.731
C05186=1018.195,165.159,-121.197,167.558,52.392,159.732
C05187=1018.191,164.910,-121.176,167.554,52.401,159.733
C05188=1018.185,164.661,-121.154,167.551,52.409,159.734
C05189=1018.180,164.412,-121.133,167.547,52.418,159.735
C05190=1018.176,164.163,-121.112,167.543,52.426,159.736
C05191=1018.171,163.913,-121.092,167.539,52.434,159.737
C05192=1018.167,163.665,-121.070,167.536,52.443,159.738
C05193=1018.161,163.416,-121.050,167.532,52.451,159.739
C05194=1018.157,163.167,-121.028,167.529,52.460,159.740
C05195=1018.152,162.917,-121.007,167.525,52.468,159.741
C05196=1018.147,162.668,-120.987,167.521,52.476,159.742
C05197=1018.142,162.419,-120.965,167.518,52.485,159.743
C05198=1018.137,162.171,-120.945,167.514,52.493,159.744
C05199=1018.133,161.922,-120.923,167.511,52.502,159.745
C05200=1018.128,161.672,-120.902,167.507,52.510,159.746
C05201=1018.123,161.423,-120.882,167.504,52.518,159.747
C05202=1018.119,161.174,-120.861,167.500,52.527,159.748
C05203=1018.114,160.925,-120.840,167.497,52.535,159.749
C05204=1018.109,160.676,-120.819,167.493,52.544,159.750
C05205=1018.104,160.427,-120.798,167.490,52.552,159.751
C05206=1018.099,160.178,-120.777,167.486,52.560,159.752
C05207=1018.096,159.929,-120.756,167.483,52.569,159.753
C05208=1018.090,159.680,-120.736,167.479,52.577,159.754
C05209=1018.086,159.430,-120.714,167.476,52.586,159.755
C05210=1018.080,159.181,-120.694,167.472,52.594,159.756
C05211=1018.077,158.933,-120.673,167.468,52.602,159.757
C05212=1018.072,158.683,-120.652,167.465,52.611,159.758
C05213=1018.067,158.434,-120.631,167.461,52.620,159.759
C05214=1018.062,158.185,-120.611,167.457,52.629,159.760
C05215=1018.056,157.936,-120.590,167.454,52.637,159.761
C05216=1018.052,157.687,-120.570,167.450,52.645,159.762
C05217=1018.047,157.438,-120.550,167.447,52.654,159.763
C05218=1018.042,157.188,-120.529,167.443,52.662,159.764
C05219=1018.037,156.939,-120.508,167.440,52.671,159.765
C05220=1018.032,156.691,-120.488,167.436,52.681,159.766
C05221=1018.027,156.441,-120.468,167.432,52.689,159.767
C05222=1018.022,156.192,-120.448,167.429,52.698,159.768
C05223=1018.017,155.943,-120.427,167.426,52.706,159.769
C05224=1018.012,155.694,-120.407,167.422,52.715,159.770
C05225=1018.007,155.412,-120.384,167.418,52.724,159.772
C05226=1018.001,155.131,-120.361,167.415,52.734,159.773
C05227=1017.995,154.849,-120.337,167.410,52.744,159.774
C05228=1017.990,154.568,-120.315,167.407,52.754,159.775
C05229=1017.985,154.319,-120.295,167.403,52.762,159.776
C05230=1017.980,154.070,-120.275,167.400,52.771,159.777
C05231=1017.975,153.820,-120.254,167.397,52.779,159.778
C05232=1017.971,153.572,-120.234,167.393,52.788,159.779
C05233=1017.966,153.322,-120.214,167.390,52.796,159.780
C05234=1017.961,153.073,-120.193,167.386,52.805,159.781
C05235=1017.956,152.824,-120.173,167.382,52.814,159.782
C05236=1017.951,152.575,-120.153,167.379,52.823,159.783
C05237=1017.946,152.326,-120.133,167.375,52.832,159.784
C05238=1017.941,152.076,-120.112,167.372,52.840,159.785
C05239=1017.936,151.827,-120.093,167.369,52.849,159.787
C05240=1017.931,151.578,-120.072,167.365,52.858,159.788
C05241=1017.926,151.328,-120.052,167.362,52.866,159.789
C05242=1017.921,151.080,-120.032,167.359,52.875,159.790
C05243=1017.917,150.830,-120.012,167.355,52.883,159.791
C05244=1017.912,150.582,-119.992,167.352,52.892,159.792
C05245=1017.907,150.332,-119.972,167.349,52.901,159.793
C05246=1017.902,150.083,-119.952,167.345,52.909,159.794
C05247=1017.897,149.834,-119.932,167.341,52.918,159.795
C05248=1017.891,149.585,-119.912,167.338,52.927,159.796
C05249=1017.886,149.335,-119.892,167.334,52.936,159.797
C05250=1017.882,149.087,-119.872,167.331,52.944,159.798
C05251=1017.877,148.837,-119.852,167.328,52.953,159.799
C05252=1017.872,148.589,-119.832,167.324,52.962,159.800
C05253=1017.867,148.339,-119.812,167.321,52.970,159.801
C05254=1017.862,148.091,-119.792,167.318,52.979,159.802
C05255=1017.858,147.841,-119.772,167.314,52.988,159.804
C05256=1017.852,147.592,-119.752,167.311,52.996,159.805
C05257=1017.848,147.343,-119.732,167.308,53.005,159.806
C05258=1017.843,147.093,-119.712,167.305,53.014,159.807
C05259=1017.838,146.845,-119.692,167.301,53.022,159.808
C05260=1017.833,146.595,-119.672,167.298,53.031,159.809
C05261=1017.828,146.347,-119.653,167.295,53.040,159.810
C05262=1017.823,146.097,-119.633,167.291,53.048,159.811
C05263=1017.818,145.847,-119.613,167.288,53.057,159.812
C05264=1017.813,145.599,-119.593,167.285,53.066,159.813
C05265=1017.808,145.349,-119.573,167.281,53.074,159.814
C05266=1017.803,145.100,-119.554,167.278,53.083,159.815
C05267=1017.798,144.851,-119.534,167.275,53.092,159.817
C05268=1017.794,144.602,-119.514,167.271,53.101,159.818
C05269=1017.789,144.352,-119.494,167.268,53.110,159.819
C05270=1017.784,144.104,-119.475,167.264,53.118,159.820
C05271=1017.779,143.854,-119.456,167.261,53.127,159.821
C05272=1017.774,143.606,-119.435,167.258,53.136,159.822
C05273=1017.768,143.356,-119.416,167.255,53.145,159.823
C05274=1017.764,143.107,-119.397,167.251,53.153,159.824
C05275=1017.759,142.857,-119.377,167.248,53.162,159.825
C05276=1017.754,142.609,-119.358,167.245,53.171,159.826
C05277=1017.749,142.359,-119.337,167.242,53.180,159.827
C05278=1017.744,142.110,-119.318,167.238,53.188,159.828
C05279=1017.739,141.861,-119.299,167.235,53.197,159.829
C05280=1017.734,141.612,-119.279,167.232,53.206,159.831
C05281=1017.729,141.362,-119.259,167.228,53.214,159.832
C05282=1017.724,141.114,-119.241,167.225,53.223,159.833
C05283=1017.719,140.864,-119.221,167.222,53.232,159.834
C05284=1017.715,140.615,-119.201,167.219,53.241,159.835
C05285=1017.709,140.366,-119.181,167.215,53.249,159.836
C05286=1017.705,140.117,-119.162,167.212,53.258,159.837
C05287=1017.700,139.867,-119.142,167.209,53.267,159.838
C05288=1017.695,139.618,-119.123,167.206,53.276,159.839
C05289=1017.689,139.337,-119.101,167.202,53.286,159.840
C05290=1017.684,139.055,-119.079,167.198,53.296,159.842
C05291=1017.679,138.774,-119.057,167.195,53.306,159.843
C05292=1017.673,138.492,-119.035,167.191,53.316,159.844
C05293=1017.668,138.242,-119.015,167.188,53.325,159.845
C05294=1017.664,137.993,-118.996,167.184,53.333,159.846
C05295=1017.658,137.744,-118.976,167.181,53.342,159.847
C05296=1017.654,137.495,-118.957,167.178,53.351,159.849
C05297=1017.649,137.246,-118.938,167.175,53.360,159.850
C05298=1017.644,136.996,-118.918,167.171,53.368,159.851
C05299=1017.639,136.748,-118.899,167.168,53.377,159.852
C05300=1017.634,136.498,-118.879,167.165,53.386,159.853
C05301=1017.629,136.249,-118.861,167.162,53.395,159.854
C05302=1017.624,136.000,-118.841,167.159,53.403,159.855
C05303=1017.618,135.751,-118.822,167.156,53.412,159.856
C05304=1017.614,135.501,-118.803,167.153,53.421,159.857
C05305=1017.609,135.252,-118.784,167.149,53.430,159.859
C05306=1017.604,135.003,-118.764,167.146,53.439,159.860
C05307=1017.599,134.754,-118.746,167.143,53.447,159.861
C05308=1017.594,134.504,-118.726,167.140,53.456,159.862
C05309=1017.589,134.255,-118.707,167.137,53.465,159.863
C05310=1017.584,134.006,-118.689,167.134,53.474,159.864
C05311=1017.580,133.756,-118.669,167.131,53.483,159.865
C05312=1017.574,133.507,-118.650,167.127,53.492,159.866
C05313=1017.569,133.259,-118.631,167.124,53.501,159.867
C05314=1017.564,133.009,-118.611,167.121,53.510,159.868
C05315=1017.560,132.760,-118.593,167.118,53.519,159.870
C05316=1017.555,132.511,-118.574,167.114,53.527,159.871
C05317=1017.550,132.261,-118.554,167.111,53.536,159.872
C05318=1017.545,132.012,-118.535,167.108,53.545,159.873
C05319=1017.540,131.763,-118.516,167.105,53.554,159.874
C05320=1017.535,131.513,-118.497,167.102,53.563,159.875
C05321=1017.530,131.264,-118.478,167.099,53.571,159.876
C05322=1017.525,131.016,-118.459,167.096,53.580,159.877
C05323=1017.520,130.767,-118.440,167.093,53.589,159.878
C05324=1017.516,130.516,-118.421,167.090,53.598,159.880
C05325=1017.511,130.268,-118.402,167.086,53.607,159.881
C05326=1017.506,130.019,-118.383,167.083,53.616,159.882
C05327=1017.501,129.769,-118.364,167.081,53.624,159.883
C05328=1017.496,129.520,-118.345,167.078,53.633,159.884
C05329=1017.492,129.270,-118.327,167.074,53.643,159.885
C05330=1017.486,129.021,-118.307,167.071,53.652,159.886
C05331=1017.481,128.771,-118.289,167.068,53.660,159.887
C05332=1017.476,128.523,-118.270,167.065,53.669,159.888
C05333=1017.471,128.273,-118.252,167.061,53.678,159.890
C05334=1017.466,128.024,-118.233,167.058,53.687,159.891
C05335=1017.461,127.775,-118.215,167.055,53.696,159.892
C05336=1017.456,127.526,-118.196,167.052,53.705,159.893
C05337=1017.450,127.276,-118.177,167.049,53.714,159.894
C05338=1017.445,127.027,-118.158,167.046,53.723,159.895
C05339=1017.441,126.778,-118.140,167.043,53.732,159.897
C05340=1017.435,126.529,-118.121,167.040,53.741,159.898
C05341=1017.430,126.279,-118.103,167.037,53.750,159.899
C05342=1017.425,126.030,-118.084,167.034,53.759,159.900
C05343=1017.420,125.781,-118.066,167.031,53.767,159.901
C05344=1017.415,125.532,-118.047,167.028,53.777,159.902
C05345=1017.410,125.282,-118.028,167.025,53.786,159.903
C05346=1017.405,125.033,-118.010,167.022,53.795,159.904
C05347=1017.400,124.784,-117.991,167.019,53.804,159.906
C05348=1017.396,124.534,-117.973,167.016,53.813,159.907
C05349=1017.391,124.286,-117.954,167.013,53.822,159.908
C05350=1017.385,124.036,-117.935,167.010,53.831,159.909
C05351=1017.380,123.787,-117.916,167.007,53.840,159.910
C05352=1017.375,123.537,-117.898,167.004,53.848,159.911
C05353=1017.369,123.256,-117.877,167.000,53.858,159.913
C05354=1017.364,122.974,-117.857,166.997,53.868,159.914
C05355=1017.358,122.692,-117.836,166.993,53.879,159.915
C05356=1017.353,122.411,-117.814,166.989,53.889,159.916
C05357=1017.348,122.162,-117.796,166.987,53.898,159.917
C05358=1017.344,121.912,-117.778,166.984,53.907,159.919
C05359=1017.338,121.663,-117.759,166.981,53.916,159.920
